	ELSIF (#coordSystem = "CS_MCS" AND #startPositionCoordSystem <> "CS_MCS")
	  OR (#coordSystem = "CS_JCS" AND #startPositionCoordSystem <> "CS_JCS")
	THEN
	  // Transform cartesian lastPos to MCS or JCS
	  #inverseKinematicsTransformation(AxesGroup         := #toKinematics,
	                                   Enable            := TRUE,
	                                   Position          := #statStartPosition,
	                                   CoordSystem       := #startPositionCoordSystem,
	                                   AxesCoordSystem   := #coordSystem,
	                                   LinkConstellation := #startLinkConstellation,
	                                   ErrorId           => #tempRetVal,
	                                   AxesPosition      => #statStartPosition);
	  
	  // check for error in last position calculation
	  IF #tempRetVal <> 16#0 THEN
	    #status := #tempRetVal;
	    RETURN;
	  END_IF;
	  
	ELSIF (#coordSystem <> "CS_MCS" AND #startPositionCoordSystem = "CS_MCS")
	  OR (#coordSystem <> "CS_JCS" AND #startPositionCoordSystem = "CS_JCS")
	THEN
	  // Transform axial lastPos to target cartesian CS
	  #kinematicsTransformation(AxesGroup         := #toKinematics,
	                            Enable            := TRUE,
	                            AxesPosition      := #statStartPosition,
	                            CoordSystem       := #coordSystem,
	                            AxesCoordSystem   := #startPositionCoordSystem,
	                            ErrorId           => #tempRetVal,
	                            Position          => #statStartPosition,
	                            LinkConstellation => #resultingLinkConstellation);
	  
	  // check for error in last position calculation
	  IF #tempRetVal <> 16#0 THEN
	    #status := #tempRetVal;
	    RETURN;
	  END_IF;
	  
	ELSE
	  // Transform Start position to correct CS 
	  "LKinCtrl_FrameTrans"(coordSystem    := #coordSystem, // Actual/Target CS
	                        coordSystemOld := #startPositionCoordSystem, // Last CS
	                        OCSFrames      := #OCSFrames, // OCS frames
	                        userFrames     := #userFrames,
	                        position       := #statStartPosition); // Position to be transformed
	END_IF;
	
	
	//------------------------------------------------------------------------------------------
	// Update linkConstellation
	//------------------------------------------------------------------------------------------
	// LinkConstellation can only be set at sPTP command in WCS/OCS
	IF #coordSystem <> "CS_MCS"
	  AND #coordSystem <> "CS_JCS"
	  AND #moveDirectParameter.linkConstellation <> 16#FFFF_FFFF
	  AND (#cmdType = "LKINCTRL_MC_MOVEDIRECTABS"
	  OR #cmdType = "LKINCTRL_MC_MOVEDIRECTREL")
	THEN
	  // LinkConstellation is changed
	  #resultingLinkConstellation := DWORD_TO_DINT(#moveDirectParameter.linkConstellation);
	END_IF;
	
	//------------------------------------------------------------------------------------------
	// Update PositionMode
	//------------------------------------------------------------------------------------------
	// PositionMode is only valid for absolute SPTP command in WCS/OCS
	IF #coordSystem <> "CS_MCS"
	  AND #moveDirectParameter.positionMode = "PM_ABS_REL" // Relative A coordinate
	  AND #cmdType = "LKINCTRL_MC_MOVEDIRECTABS"
	THEN
	  // Calc correct orientation position
	    #resultingPosition[4] := #statStartPosition[4] + #statCommandPosition[4];
	  //#statCommandPosition[4] := #resultingPosition[4]; // update tempPosition
	    ;
	END_IF;
	
	//------------------------------------------------------------------------------------------
	// ParameterValid bit check -> Check if all positions are valid -> LKinLang mechanism
	//------------------------------------------------------------------------------------------
	CASE #cmdType OF
	  "LKINCTRL_MC_MOVELINEARABS", "LKINCTRL_MC_MOVECIRCULARABS", "LKINCTRL_MC_MOVEDIRECTABS", "LKINCTRL_MC_MOVELINEARPICKANDPLACE":  // Absolute commands
	    FOR #tempIndex := 1 TO "LKINCTRL_NO_OF_VALID_BITS" DO
	      // Check valid bits and copy last pos (X,Y,Z,A) where missing
	      IF #parameterValid[#tempIndex] = FALSE THEN
	        #statCommandPosition[#tempIndex] := #statStartPosition[#tempIndex]; // write lastPos as target pos if invalid
	      ELSE
	        CONTINUE;
	      END_IF;
	    END_FOR;
	    
	  "LKINCTRL_MC_MOVELINEARREL", "LKINCTRL_MC_MOVECIRCULARREL", "LKINCTRL_MC_MOVEDIRECTREL":  // Relative commands
	    FOR #tempIndex := 1 TO "LKINCTRL_NO_OF_VALID_BITS" DO
	      // Check valid bits and set absolute pos to 0.0 (X,Y,Z,A)
	      IF #parameterValid[#tempIndex] = FALSE THEN
	        #statCommandPosition[#tempIndex] := 0.0; // write no increment as relative target pos if invalid
	      ELSE
	        CONTINUE;
	      END_IF;
	    END_FOR;
	    
	  ELSE  // Nothing to do for this cmdType
	    ;
	END_CASE;
	
	//------------------------------------------------------------------------------------------
	// Convert circle mode 3 (Gcode notation) to circle mode 1 (arc + endPoint)
	//------------------------------------------------------------------------------------------
	// --> CmdType = 3 (always absolute as result)
	// --> CircleParameters = calculated arc, updated auxPoint, circMode 1
	IF #circleParameters.circMode = "LKINCTRL_CIRCMODE_GCODE" THEN
	  #tempRetVal := "LKinCtrl_ConvCircMode3To1"(coordinates := #statCommandPosition,
	                                             startPosition := #statStartPosition,
	                                             cmdType := #cmdType,
	                                             circleParameters := #circleParameters);
	  
	  // check for error in circle calculation
	  IF #tempRetVal <> 16#0 THEN
	    #status := #tempRetVal;
	    RETURN;
	  END_IF;
	END_IF;
	
	//------------------------------------------------------------------------------------------
	// Handle relative shift
	//------------------------------------------------------------------------------------------
	IF #relativeShift.shiftActive = TRUE
	  AND #relativeShift.coordinateSystem = #coordSystem
	THEN
	  IF #cmdType = "LKINCTRL_MC_MOVELINEARABS"
	    OR #cmdType = "LKINCTRL_MC_MOVEDIRECTABS"
	    OR #cmdType = "LKINCTRL_MC_MOVECIRCULARABS"
	    OR #cmdType = "LKINCTRL_MC_MOVELINEARPICKANDPLACE"
	  THEN
	    // Translation and rotation (end point)
	    "LKinCtrl_OcsToWcs"(ocsX      := #relativeShift.coordinates[1],
	                        ocsY      := #relativeShift.coordinates[2],
	                        ocsZ      := #relativeShift.coordinates[3],
	                        ocsA      := #relativeShift.coordinates[4],
	                        ocsB      := #relativeShift.coordinates[5],
	                        ocsC      := #relativeShift.coordinates[6],
	                        pointXOcs := #statCommandPosition[1],
	                        pointYOcs := #statCommandPosition[2],
	                        pointZOcs := #statCommandPosition[3],
	                        pointAOcs := #statCommandPosition[4],
	                        pointBOcs := #statCommandPosition[5],
	                        pointCOcs := #statCommandPosition[6],
	                        pointXWcs => #statCommandPosition[1],
	                        pointYWcs => #statCommandPosition[2],
	                        pointZWcs => #statCommandPosition[3],
	                        pointAWcs => #statCommandPosition[4],
	                        pointBWcs => #statCommandPosition[5],
	                        pointCWcs => #statCommandPosition[6]);
	    
	    // Translation and rotation (aux point)
	    "LKinCtrl_OcsToWcs"(ocsX      := #relativeShift.coordinates[1],
	                        ocsY      := #relativeShift.coordinates[2],
	                        ocsZ      := #relativeShift.coordinates[3],
	                        ocsA      := #relativeShift.coordinates[4],
	                        ocsB      := #relativeShift.coordinates[5],
	                        ocsC      := #relativeShift.coordinates[6],
	                        pointXOcs := #circleParameters.auxPoint[1],
	                        pointYOcs := #circleParameters.auxPoint[2],
	                        pointZOcs := #circleParameters.auxPoint[3],
	                        pointAOcs := 0.0,
	                        pointBOcs := 0.0,
	                        pointCOcs := 0.0,
	                        pointXWcs => #circleParameters.auxPoint[1],
	                        pointYWcs => #circleParameters.auxPoint[2],
	                        pointZWcs => #circleParameters.auxPoint[3],
	                        pointAWcs => #tempAuxPoint[4],
	                        pointBWcs => #tempAuxPoint[5],
	                        pointCWcs => #tempAuxPoint[6]);
	    
	  ELSIF #cmdType = "LKINCTRL_MC_MOVELINEARREL"
	    OR #cmdType = "LKINCTRL_MC_MOVEDIRECTREL"
	    OR #cmdType = "LKINCTRL_MC_MOVECIRCULARREL"
	  THEN
	    // Only rotation (end point)
	    "LKinCtrl_OcsToWcs"(ocsX      := 0.0,
	                        ocsY      := 0.0,
	                        ocsZ      := 0.0,
	                        ocsA      := #relativeShift.coordinates[4],
	                        ocsB      := #relativeShift.coordinates[5],
	                        ocsC      := #relativeShift.coordinates[6],
	                        pointXOcs := #statCommandPosition[1],
	                        pointYOcs := #statCommandPosition[2],
	                        pointZOcs := #statCommandPosition[3],
	                        pointAOcs := 0.0,
	                        pointBOcs := 0.0,
	                        pointCOcs := 0.0,
	                        pointXWcs => #statCommandPosition[1],
	                        pointYWcs => #statCommandPosition[2],
	                        pointZWcs => #statCommandPosition[3],
	                        pointAWcs => #tempAuxPoint[4],
	                        pointBWcs => #tempAuxPoint[5],
	                        pointCWcs => #tempAuxPoint[6]);
	    
	    // Only rotation (aux point)
	    "LKinCtrl_OcsToWcs"(ocsX      := 0.0,
	                        ocsY      := 0.0,
	                        ocsZ      := 0.0,
	                        ocsA      := #relativeShift.coordinates[4],
	                        ocsB      := #relativeShift.coordinates[5],
	                        ocsC      := #relativeShift.coordinates[6],
	                        pointXOcs := #circleParameters.auxPoint[1],
	                        pointYOcs := #circleParameters.auxPoint[2],
	                        pointZOcs := #circleParameters.auxPoint[3],
	                        pointAOcs := 0.0,
	                        pointBOcs := 0.0,
	                        pointCOcs := 0.0,
	                        pointXWcs => #circleParameters.auxPoint[1],
	                        pointYWcs => #circleParameters.auxPoint[2],
	                        pointZWcs => #circleParameters.auxPoint[3],
	                        pointAWcs => #tempAuxPoint[4],
	                        pointBWcs => #tempAuxPoint[5],
	                        pointCWcs => #tempAuxPoint[6]);
	  ELSE
	    ;// No calculation necessary
	  END_IF;
	END_IF;
	
	//------------------------------------------------------------------------------------------
	// Calculate resulting absoulte position
	//------------------------------------------------------------------------------------------
	#tempRetVal := "LKinCtrl_CalcResultingPos"(cmdType := #cmdType,
	                                           cartesianPos := #statCommandPosition,
	                                           circleParameters := #circleParameters,
	                                           startPosition := #statStartPosition,
	                                           commandLengthIsZero => #cmdLengthZero,
	                                           resultingDistance => #resultingDistance,
	                                           resultingPosition => #resultingPosition,
	                                           resultingAuxPoint => #resultingAuxPoint);  
	
	// check for error in resulting position calculation
	IF #tempRetVal <> 16#0 THEN
	  #status := #tempRetVal;
	  RETURN;
	END_IF;
	
	//------------------------------------------------------------------------------------------
	// Transform UCS commands into WCS
	// At this point all coordinates are calauclated in UCS -> Transform them in WCS to be able to execute system commands
	//------------------------------------------------------------------------------------------
	IF #coordSystem >= "LKINCTRL_CS_NO_OF_FIRST_USER_FRAME"
	  AND #coordSystem <= "LKINCTRL_CS_NO_OF_LAST_USER_FRAME"
	THEN
	  CASE #cmdType OF
	    "LKINCTRL_MC_MOVELINEARABS", "LKINCTRL_MC_MOVECIRCULARABS", "LKINCTRL_MC_MOVEDIRECTABS",  // Absolute commands
	    "LKINCTRL_MC_MOVELINEARREL", "LKINCTRL_MC_MOVECIRCULARREL", "LKINCTRL_MC_MOVEDIRECTREL":  // Relative commands
	      // Up to this point all positions (start, resulting & distance) are in UCS
	      // --> Calculate new values in WCS
	      
	      // Transform start position into WCS
	      "LKinCtrl_OcsToWcs"(ocsX      := #userFrames[#coordSystem].x,
	                          ocsY      := #userFrames[#coordSystem].y,
	                          ocsZ      := #userFrames[#coordSystem].z,
	                          ocsA      := #userFrames[#coordSystem].a,
	                          ocsB      := #userFrames[#coordSystem].b,
	                          ocsC      := #userFrames[#coordSystem].c,
	                          pointXOcs := #statStartPosition[1],
	                          pointYOcs := #statStartPosition[2],
	                          pointZOcs := #statStartPosition[3],
	                          pointAOcs := #statStartPosition[4],
	                          pointBOcs := #statStartPosition[5],
	                          pointCOcs := #statStartPosition[6],
	                          pointXWcs => #statStartPosition[1],
	                          pointYWcs => #statStartPosition[2],
	                          pointZWcs => #statStartPosition[3],
	                          pointAWcs => #statStartPosition[4],
	                          pointBWcs => #statStartPosition[5],
	                          pointCWcs => #statStartPosition[6]);
	      
	      // Transform resulting position into WCS
	      "LKinCtrl_OcsToWcs"(ocsX      := #userFrames[#coordSystem].x,
	                          ocsY      := #userFrames[#coordSystem].y,
	                          ocsZ      := #userFrames[#coordSystem].z,
	                          ocsA      := #userFrames[#coordSystem].a,
	                          ocsB      := #userFrames[#coordSystem].b,
	                          ocsC      := #userFrames[#coordSystem].c,
	                          pointXOcs := #resultingPosition[1],
	                          pointYOcs := #resultingPosition[2],
	                          pointZOcs := #resultingPosition[3],
	                          pointAOcs := #resultingPosition[4],
	                          pointBOcs := #resultingPosition[5],
	                          pointCOcs := #resultingPosition[6],
	                          pointXWcs => #resultingPosition[1],
	                          pointYWcs => #resultingPosition[2],
	                          pointZWcs => #resultingPosition[3],
	                          pointAWcs => #resultingPosition[4],
	                          pointBWcs => #resultingPosition[5],
	                          pointCWcs => #resultingPosition[6]);
	      
	      // Transform resulting aux position into WCS
	      "LKinCtrl_OcsToWcs"(ocsX      := #userFrames[#coordSystem].x,
	                          ocsY      := #userFrames[#coordSystem].y,
	                          ocsZ      := #userFrames[#coordSystem].z,
	                          ocsA      := #userFrames[#coordSystem].a,
	                          ocsB      := #userFrames[#coordSystem].b,
	                          ocsC      := #userFrames[#coordSystem].c,
	                          pointXOcs := #resultingAuxPoint[1],
	                          pointYOcs := #resultingAuxPoint[2],
	                          pointZOcs := #resultingAuxPoint[3],
	                          pointAOcs := 0,
	                          pointBOcs := 0,
	                          pointCOcs := 0,
	                          pointXWcs => #resultingAuxPoint[1],
	                          pointYWcs => #resultingAuxPoint[2],
	                          pointZWcs => #resultingAuxPoint[3],
	                          pointAWcs => #tempAuxPoint[4],
	                          pointBWcs => #tempAuxPoint[5],
	                          pointCWcs => #tempAuxPoint[6]);
	      
	      // Calc resulting distance in WCS
	      FOR #tempIndex := 1 TO 6 DO
	        #resultingDistance[#tempIndex] := #resultingPosition[#tempIndex] - #statStartPosition[#tempIndex];
	      END_FOR;
	      
	      #coordSystem := "CS_WCS"; // Set CS to WCS
	  END_CASE;
	END_IF;
	
	
	
	
	
END_FUNCTION_BLOCK

FUNCTION "LKinCtrl_FrameTrans" : Void
TITLE = LKinCtrl_FrameTrans
{ S7_Optimized_Access := 'TRUE' }
AUTHOR : 'handling.team.automation@siemens.com'
FAMILY : LKinCtrl
VERSION : 5.0
//Transform postion into different coordinate systems
   VAR_INPUT 
      coordSystem : DInt;   // target coordinate system
      coordSystemOld : DInt;   // previous coordinate system
      OCSFrames : Array[1..3] of "LKinCtrl_typeFrame";   // OCS frames
      userFrames : Array["LKINCTRL_CS_NO_OF_FIRST_USER_FRAME".."LKINCTRL_CS_NO_OF_LAST_USER_FRAME"] of "LKinCtrl_typeFrame";   // User frames
   END_VAR

   VAR_IN_OUT 
      position : Array[1..6] of LReal;   // position to be transformed
   END_VAR


BEGIN
	//==========================================================================================
	// SIEMENS AG
	// (c)Copyright 2020 All Rights Reserved
	//------------------------------------------------------------------------------------------
	// Library: LKinCtrl
	// Tested with: S7-1517T-3 PN/DP
	// Engineering: TIA Portal V15
	// Restrictions: ---
	// Requirements: S7-1500T FW 2.5
	// Functionality: LKinCtrl_FrameTrans
	// The FC calculates a given position transformed into or from another coordinate system
	// depending on the actual / previous coordinate system of the cmd
	//
	// Support: tech.team.motioncontrol@siemens.com
	// Note: Parameter comments are only available in language 'English (United States)'
	//------------------------------------------------------------------------------------------
	// Change log table:
	// Version    Date          Expert in charge    Changes applied
	// 01.00.00   16.04.2019    JR                  First release version v1.0
	// 02.00.00   14.04.2020    FR                  Use array of frames
	// 03.00.00   18.01.2022    FR                  Update to 6 axis
	//===========================================================================================
	
	// Check if last CS differs from actual CS
	IF #coordSystem = #coordSystemOld THEN
	  // No calculation needed --> Return
	  RETURN;
	END_IF;
	
	// Calc new position
	// =================
	// Check if last CS was a OCS
	// YES: Transform position to WCS
	// NO: Do nothing --> Position is already in WCS
	CASE #coordSystemOld OF
	  "CS_OCS1".."CS_OCS3": // OCS
	    "LKinCtrl_OcsToWcs"(ocsX      := #OCSFrames[#coordSystemOld].x,
	                        ocsY      := #OCSFrames[#coordSystemOld].y,
	                        ocsZ      := #OCSFrames[#coordSystemOld].z,
	                        ocsA      := #OCSFrames[#coordSystemOld].a,
	                        ocsB      := #OCSFrames[#coordSystemOld].b,
	                        ocsC      := #OCSFrames[#coordSystemOld].c,
	                        pointXOcs := #position[1],
	                        pointYOcs := #position[2],
	                        pointZOcs := #position[3],
	                        pointAOcs := #position[4],
	                        pointBOcs := #position[5],
	                        pointCOcs := #position[6],
	                        pointXWcs => #position[1],
	                        pointYWcs => #position[2],
	                        pointZWcs => #position[3],
	                        pointAWcs => #position[4],
	                        pointBWcs => #position[5],
	                        pointCWcs => #position[6]);
	    
	  "LKINCTRL_CS_NO_OF_FIRST_USER_FRAME".."LKINCTRL_CS_NO_OF_LAST_USER_FRAME":  // User frame
	    "LKinCtrl_OcsToWcs"(ocsX      := #userFrames[#coordSystemOld].x,
	                        ocsY      := #userFrames[#coordSystemOld].y,
	                        ocsZ      := #userFrames[#coordSystemOld].z,
	                        ocsA      := #userFrames[#coordSystemOld].a,
	                        ocsB      := #userFrames[#coordSystemOld].b,
	                        ocsC      := #userFrames[#coordSystemOld].c,
	                        pointXOcs := #position[1],
	                        pointYOcs := #position[2],
	                        pointZOcs := #position[3],
	                        pointAOcs := #position[4],
	                        pointBOcs := #position[5],
	                        pointCOcs := #position[6],
	                        pointXWcs => #position[1],
	                        pointYWcs => #position[2],
	                        pointZWcs => #position[3],
	                        pointAWcs => #position[4],
	                        pointBWcs => #position[5],
	                        pointCWcs => #position[6]);
	    
	  ELSE
	    ;
	END_CASE;
	
	
	// Check if target CS is a OCS
	// YES: Transform position to target OCS
	// NO: Target CS is WCS --> Position is already in WCS from above
	CASE #coordSystem OF
	  "CS_OCS1".."CS_OCS3": // OCS
	    "LKinCtrl_WcsToOcs"(ocsX      := #OCSFrames[#coordSystem].x,
	                        ocsY      := #OCSFrames[#coordSystem].y,
	                        ocsZ      := #OCSFrames[#coordSystem].z,
	                        ocsA      := #OCSFrames[#coordSystem].a,
	                        ocsB      := #OCSFrames[#coordSystem].b,
	                        ocsC      := #OCSFrames[#coordSystem].c,
	                        pointXWcs := #position[1],
	                        pointYWcs := #position[2],
	                        pointZWcs := #position[3],
	                        pointAWcs := #position[4],
	                        pointBWcs := #position[5],
	                        pointCWcs := #position[6],
	                        pointXOcs => #position[1],
	                        pointYOcs => #position[2],
	                        pointZOcs => #position[3],
	                        pointAOcs => #position[4],
	                        pointBOcs => #position[5],
	                        pointCOcs => #position[6]);
	    
	  "LKINCTRL_CS_NO_OF_FIRST_USER_FRAME".."LKINCTRL_CS_NO_OF_LAST_USER_FRAME":  // User frame
	    "LKinCtrl_WcsToOcs"(ocsX      := #userFrames[#coordSystem].x,
	                        ocsY      := #userFrames[#coordSystem].y,
	                        ocsZ      := #userFrames[#coordSystem].z,
	                        ocsA      := #userFrames[#coordSystem].a,
	                        ocsB      := #userFrames[#coordSystem].b,
	                        ocsC      := #userFrames[#coordSystem].c,
	                        pointXWcs := #position[1],
	                        pointYWcs := #position[2],
	                        pointZWcs := #position[3],
	                        pointAWcs := #position[4],
	                        pointBWcs := #position[5],
	                        pointCWcs := #position[6],
	                        pointXOcs => #position[1],
	                        pointYOcs => #position[2],
	                        pointZOcs => #position[3],
	                        pointAOcs => #position[4],
	                        pointBOcs => #position[5],
	                        pointCOcs => #position[6]);
	    
	  ELSE
	    ;
	END_CASE;
	
	
	
END_FUNCTION

FUNCTION "LKinCtrl_ConvCircMode3To1" : Word
TITLE = LKinCtrl_ConvCircMode3To1
{ S7_Optimized_Access := 'TRUE' }
AUTHOR : 'handling.team.automation@siemens.com'
FAMILY : LKinCtrl
VERSION : 5.0
//The FC converts a circular motion command programmed with circMode 3 (GCode) to a circular command programmed with circMode 1 (center point and arc given)
   VAR_INPUT 
      coordinates : Array[1..6] of LReal;   // endPoint from path data element
      startPosition : Array[1..6] of LReal;
   END_VAR

   VAR_IN_OUT 
      cmdType : Int;   // cmdType of path data element
      circleParameters : "LKinCtrl_typeCircleParameters";   // circle parameters of path data element
   END_VAR

   VAR_TEMP 
      tempAuxPoint : Array[1..3] of LReal;   // resulting auxPoint
      tempEndPointResult : Array[1..6] of LReal;   // resulting endPoint
      tempOM : Array[1..2] of LReal;   // temporary math variable
      tempMS : Array[1..2] of LReal;   // temporary math variable
      tempME : Array[1..2] of LReal;   // temporary math variable
      tempAxisVector : Array[1..2] of LReal;   // temporary math variable
      tempScalarProd_ME_Axis : LReal;   // temporary math variable
      tempScalarProd_MS_Axis : LReal;   // temporary math variable
      tempLength_ME : LReal;   // temporary math variable
      tempLength_MS : LReal;   // temporary math variable
      tempAngleME_rad : LReal;   // temporary math variable
      tempAngleMS_rad : LReal;   // temporary math variable
      tempAngleME_deg : LReal;   // temporary math variable
      tempAngleMS_deg : LReal;   // temporary math variable
      tempAngleDiff_deg : LReal;   // temporary math variable
      tempCtr : Int;   // temporary counter
      tempCoordinates : Array[1..6] of LReal;   // temporary array for input end point
   END_VAR

   VAR CONSTANT 
      ARC_TOLERANCE : LReal := 1.0E-09;   // Tolerance when deciding arc
      RADIUS_TOLERANCE : LReal := 0.1;   // Tolerance when comparing calculated radius
      ERR_INVALID_RADIUS : Word := 16#8201;   // Error calculated radius is invalid
   END_VAR


BEGIN
	//==========================================================================================
	// SIEMENS AG
	// (c)Copyright 2020 All Rights Reserved
	//------------------------------------------------------------------------------------------
	// Library: LKinCtrl
	// Tested with: S7-1517T-3 PN/DP
	// Engineering: TIA Portal V15
	// Restrictions: ---
	// Requirements: S7-1500T FW 2.5
	// Functionality: LKinCtrl_ConvCircMode3To1
	// The FC converts a circular motion command programmed with circMode 3 (GCode) to a circular
	// command programmed with circMode 1 (center point and arc given)
	//
	// Support: tech.team.motioncontrol@siemens.com
	// Note: Parameter comments are only available in language 'English (United States)'
	//------------------------------------------------------------------------------------------
	// Change log table:
	// Version    Date          Expert in charge    Changes applied
	// 01.00.00   03.07.2019    JR                  First release version v1.0
	// 02.00.00   06.04.2020    FR                  Changed interface to fit PathDataPreBuf and normal element
	// 02.00.01   14.01.2021    FR                  Added tolerance when calculating arc
	// 02.00.02   19.10.2021    FR                  Changed check for ACOS to allow 0.0
	// 03.00.00   18.01.2022    FR                  Update to 6 axis; Check radius for plausability
	//===========================================================================================
	
	// Init retrun value
	#LKinCtrl_ConvCircMode3To1 := 16#0;
	
	// add conversion of circMode CM: 3 circular cmds -> CM: 1
	IF (#cmdType = "LKINCTRL_MC_MOVECIRCULARABS" OR #cmdType = "LKINCTRL_MC_MOVECIRCULARREL")
	  AND #circleParameters.circMode = "LKINCTRL_CIRCMODE_GCODE"
	THEN
	  // Copy input
	  #tempCoordinates := #coordinates;
	  
	  // conversion relative to absoulte for auxPoint (and EndPoint)
	  FOR #tempCtr := 1 TO 3 DO
	    // always convert auxPoint ==> always relative in this circle definition
	    #tempAuxPoint[#tempCtr] := #startPosition[#tempCtr] + #circleParameters.auxPoint[#tempCtr];// add new auxPoint as incremental value to last position
	    #circleParameters.auxPoint[#tempCtr] := #tempAuxPoint[#tempCtr]; // copy edited auxPoint to command for later use
	  END_FOR;
	  
	  // only convert endPoint in case of relative command
	  IF #cmdType = "LKINCTRL_MC_MOVECIRCULARREL" THEN
	    #tempEndPointResult[1] := #startPosition[1] + #tempCoordinates[1];
	    #tempEndPointResult[2] := #startPosition[2] + #tempCoordinates[2];
	    #tempEndPointResult[3] := #startPosition[3] + #tempCoordinates[3];
	    #tempEndPointResult[4] := #startPosition[4] + #tempCoordinates[4];
	    #tempEndPointResult[5] := #startPosition[5] + #tempCoordinates[5];
	    #tempEndPointResult[6] := #startPosition[6] + #tempCoordinates[6];
	    #cmdType := "LKINCTRL_MC_MOVECIRCULARABS";
	  ELSE
	    #tempEndPointResult := #tempCoordinates;
	  END_IF;
	  
	  // change circMode = 3 (define center and endPoint) to circMode = 1 (define center and arc)
	  #circleParameters.circMode := "CM_CENTER";
	  
	  // ----------------------------------------------------------------
	  // different behavior for different circlePlanes - write input vectors to calc variables 2D
	  // ----------------------------------------------------------------
	  // 0: ciclePlane XZ
	  IF #circleParameters.circlePlane = "CP_XZ" THEN
	    
	    // vector origin to circle center point 
	    #tempOM[1] := #tempAuxPoint[1];
	    #tempOM[2] := #tempAuxPoint[3];
	    
	    // unit vector x axis
	    #tempAxisVector[1] := 1;
	    #tempAxisVector[2] := 0;
	    
	    // vector circle center point to start point
	    #tempMS[1] := #startPosition[1] - #tempOM[1];
	    #tempMS[2] := #tempOM[2] - #startPosition[3];
	    
	    // vector circle center point to end point
	    #tempME[1] := #tempEndPointResult[1] - #tempOM[1];
	    #tempME[2] := #tempOM[2] - #tempEndPointResult[3];
	    
	    // 1: ciclePlane YZ
	  ELSIF #circleParameters.circlePlane = "CP_YZ" THEN
	    
	    // vector origin to circle center point 
	    #tempOM[1] := #tempAuxPoint[2];
	    #tempOM[2] := #tempAuxPoint[3];
	    
	    // unit vector x axis ==> simulating y axis here due to moved commands
	    #tempAxisVector[1] := 1;
	    #tempAxisVector[2] := 0;
	    
	    // vector circle center point to start point
	    #tempMS[1] := #startPosition[2] - #tempOM[1];
	    #tempMS[2] := #startPosition[3] - #tempOM[2];
	    
	    // vector circle center point to end point
	    #tempME[1] := #tempEndPointResult[2] - #tempOM[1];
	    #tempME[2] := #tempEndPointResult[3] - #tempOM[2];
	    
	    // 2: ciclePlane XY
	  ELSIF #circleParameters.circlePlane = "CP_XY" THEN
	    
	    // vector origin to circle center point 
	    #tempOM[1] := #tempAuxPoint[1];
	    #tempOM[2] := #tempAuxPoint[2];
	    
	    // unit vector x axis
	    #tempAxisVector[1] := 1;
	    #tempAxisVector[2] := 0;
	    
	    
	    // vector circle center point to start point
	    #tempMS[1] := #startPosition[1] - #tempOM[1];
	    #tempMS[2] := #startPosition[2] - #tempOM[2];
	    
	    // vector circle center point to end point
	    #tempME[1] := #tempEndPointResult[1] - #tempOM[1];
	    #tempME[2] := #tempEndPointResult[2] - #tempOM[2];
	    
	  ELSE
	    // error ==> wrong circlePlane
	    ;
	  END_IF;
	  
	  // ----------------------------------------------------------------
	  // VECTOR CALCULATIONS
	  // ----------------------------------------------------------------
	  // calc scalar product of ME (circle center point to end point) with x axis
	  #tempScalarProd_ME_Axis := "LKinCtrl_VecScalarProd_2D"(vIn1 := #tempME, vIn2 := #tempAxisVector);
	  // calc scalar product of MS (circle center point to start point / LastPos) with x axis
	  #tempScalarProd_MS_Axis := "LKinCtrl_VecScalarProd_2D"(vIn1 := #tempMS, vIn2 := #tempAxisVector);
	  
	  // calc vector length ME
	  #tempLength_ME := "LKinCtrl_VecAbs_2D"(#tempME);
	  // calc vector length MS
	  #tempLength_MS := "LKinCtrl_VecAbs_2D"(#tempMS);
	  
	  // Check if both radius are equal
	  IF ABS(#tempLength_ME - #tempLength_MS) > #RADIUS_TOLERANCE THEN
	    #LKinCtrl_ConvCircMode3To1 := #ERR_INVALID_RADIUS;
	    RETURN;
	  END_IF;
	  
	  // calc angle ME to axis
	  #tempAngleME_rad := ACOS(#tempScalarProd_ME_Axis / (#tempLength_ME * 1));
	  
	  IF #tempME[2] < 0 THEN
	    // invert angle due to ACOS range (only 0..PI)
	    #tempAngleME_rad := 2 * "LKINCTRL_PI" - #tempAngleME_rad;
	  ELSE
	    ;
	  END_IF;
	  // convert to degrees
	  #tempAngleME_deg := #tempAngleME_rad * 180 / "LKINCTRL_PI";
	  
	  // calc angle MS to axis
	  #tempAngleMS_rad := ACOS(#tempScalarProd_MS_Axis / (#tempLength_MS * 1));
	  // check for vector Ms to point downwards (below ! (x) axis)
	  IF #tempMS[2] < 0 THEN
	    // invert angle due to ACOS range
	    #tempAngleMS_rad := 2 * "LKINCTRL_PI" - #tempAngleMS_rad;
	  ELSE
	    ;
	  END_IF;
	  // convert to degrees
	  #tempAngleMS_deg := #tempAngleMS_rad * 180 / "LKINCTRL_PI";
	  
	  
	  // ----------------------------------------------------------------
	  // separation of path choice for angle calculation
	  // ----------------------------------------------------------------
	  // 0: CCW - counterclockwise / mathematical positive angle
	  IF #circleParameters.pathChoice = "PC_POSITIVE" THEN
	    // calculate difference angle
	    #tempAngleDiff_deg := #tempAngleME_deg - #tempAngleMS_deg;
	    IF #tempAngleDiff_deg > #ARC_TOLERANCE THEN
	      // write caclulated angle
	      #circleParameters.arc := #tempAngleDiff_deg;
	    ELSE
	      // write caclulated angle ==> add 360 degrees to get positive angle value
	      #circleParameters.arc := #tempAngleDiff_deg + 360;
	    END_IF;
	    
	    // 1: CW - clockwise / mathematical negative angle
	  ELSIF #circleParameters.pathChoice = "PC_NEGATIVE" THEN
	    // calculate difference angle
	    #tempAngleDiff_deg := #tempAngleMS_deg - #tempAngleME_deg;
	    IF #tempAngleDiff_deg > #ARC_TOLERANCE THEN
	      // write caclulated angle
	      #circleParameters.arc := #tempAngleDiff_deg;
	    ELSE
	      // write caclulated angle ==> add 360 degrees to get positive angle value
	      #circleParameters.arc := #tempAngleDiff_deg + 360;
	    END_IF;
	    
	  ELSE
	    // wrong input for pathChoice
	    ;
	  END_IF;
	  
	ELSE
	  ;// nothing to do
	END_IF;
END_FUNCTION

FUNCTION "LKinCtrl_VecScalarProd_2D" : LReal
TITLE = LKinCtrl_VecScalarProd_2D
{ S7_Optimized_Access := 'TRUE' }
AUTHOR : 'handling.team.automation@siemens.com'
FAMILY : LKinCtrl
VERSION : 5.0
//Calculates the scalar product of given vectors
   VAR_INPUT 
      vIn1 : Array[1..2] of LReal;   // Input vector 1
      vIn2 : Array[1..2] of LReal;   // Input vector 2
   END_VAR


BEGIN
	//=============================================================================
	// SIEMENS AG
	// (c)Copyright 2019 All Rights Reserved
	//-----------------------------------------------------------------------------
	// Library: - 
	// Tested with: S7-1516T-3 PN
	// Engineering: TIA Portal V15
	// Restrictions: -
	// Requirements: S7-1500/S7-1500T FW 2.5
	// Functionality: Scalar product of two coordinates
	//-----------------------------------------------------------------------------
	// Change log table:
	// Version  Date       Expert in charge Changes applied
	// 01.00.00 27.08.2018 SF               created
	// 01.00.01 29.01.2019 JR               adaptions for LKinCtrl 
	//=============================================================================
	
	#LKinCtrl_VecScalarProd_2D := (* #vIn1[0]*#vIn2[0] + *)#vIn1[1] * #vIn2[1] + #vIn1[2] * #vIn2[2];
END_FUNCTION

FUNCTION "LKinCtrl_VecAbs_2D" : LReal
TITLE = LKinCtrl_VecAbs_2D
{ S7_Optimized_Access := 'TRUE' }
AUTHOR : 'handling.team.automation@siemens.com'
FAMILY : LKinCtrl
VERSION : 5.0
//Calculates the length of a given vector in 2D
   VAR_INPUT 
      vIn : Array[1..2] of LReal;   // Input vector
   END_VAR


BEGIN
	//=============================================================================
	// SIEMENS AG
	// (c)Copyright 2019 All Rights Reserved
	//-----------------------------------------------------------------------------
	// Library: - 
	// Tested with: S7-1516T-3 PN
	// Engineering: TIA Portal V15
	// Restrictions: -
	// Requirements: S7-1500/S7-1500T FW 2.5
	// Functionality: Calculate length of vector
	//-----------------------------------------------------------------------------
	// Change log table:
	// Version  Date       Expert in charge Changes applied
	// 01.00.00 27.08.2018 SF               created
	// 01.00.01 29.01.2019 JR               adaptions for LKinCtrl 
	//=============================================================================
	
	#LKinCtrl_VecAbs_2D := SQRT((* #vIn[0]*#vIn[0] + *)#vIn[1] * #vIn[1] + #vIn[2] * #vIn[2]);
END_FUNCTION

FUNCTION "LKinCtrl_CalcResultingPos" : Word
TITLE = LKinCtrl_CalcResultingPos
{ S7_Optimized_Access := 'TRUE' }
AUTHOR : 'handling.team.automation@siemens.com'
FAMILY : LKinCtrl
VERSION : 5.0
//The FC calculates the resulting last position after a given command being executed starting from a given 'previous' last position 
   VAR_INPUT 
      cmdType : Int;   // command type
      cartesianPos : Array[1..6] of LReal;   // cartesian position (target from command)
      circleParameters : "LKinCtrl_typeCircleParameters";   // circle parameters
      startPosition : Array[1..6] of LReal;   // start of command (last target position)
   END_VAR

   VAR_OUTPUT 
      commandLengthIsZero : Bool;   // TRUE: command has a length of 0.0; FALSE: Command has a length
      resultingPosition : Array[1..6] of LReal;   // resulting last position
      resultingDistance : Array[1..6] of LReal;   // distance between start and endpoint for relative commands
      resultingAuxPoint : Array[1..3] of LReal;   // resulting auxPoint
   END_VAR

   VAR_TEMP 
      tempIndex : Int;   // temporary counter
      tempCartesianPos : Array[1..6] of LReal;   // temporary copy of cartesian position (target from command)
      tempResultingAuxPoint : Array[1..3] of LReal;   // temporary resulting auxPoint
   END_VAR

   VAR CONSTANT 
      STATUS_NO_ERROR : Word := 16#0000;   // status no error occured
   END_VAR


BEGIN
	//==========================================================================================
	// SIEMENS AG
	// (c)Copyright 2020 All Rights Reserved
	//------------------------------------------------------------------------------------------
	// Library: LKinCtrl
	// Tested with: S7-1517T-3 PN/DP
	// Engineering: TIA Portal V16
	// Restrictions: ---
	// Requirements: S7-1500T FW 2.8
	// Functionality: LKinCtrl_CalcResultingPos
	// The FC calculates the resulting last position after a given command being executed
	// starting from a given 'previous' last position 
	//
	// Support: tech.team.motioncontrol@siemens.com
	// Note: Parameter comments are only available in language 'English (United States)'
	//------------------------------------------------------------------------------------------
	// Change log table:
	// Version    Date          Expert in charge    Changes applied
	// 01.00.00   11.03.2019    JR                  First release version v1.0
	// 01.00.01   17.05.2019    JR                  formal code changes fitting to styleguide
	// 02.00.00   06.04.2020    FR                  Changed interface to fit PathDataPreBuf and normal element; Also updated the calculation
	// 02.01.00   16.04.2020    FR                  Added moveDirect
	// 03.00.00   25.01.2021    FR                  Changed interface and rework
	// 04.00.00   18.01.2022    FR                  Update to 6 axis, added distance
	// 04.01.00   16.10.2023    AH                  Added relative shift
	// 04.01.00   09.01.2024    SF                  Added PickAndPlace command#
	// 04.01.01   25.04.2024    JH                  Bugfix for uninitialized output
	// 04.02.00   11.07.2024    AH                  Fixed wrong calculation of circularCommand in UCS
	//===========================================================================================
	
	// ---------------------------------------------------------
	// Initialize return value to no error
	// ---------------------------------------------------------
	#LKinCtrl_CalcResultingPos := #STATUS_NO_ERROR;
	#commandLengthIsZero := FALSE;
	
	// ---------------------------------------------------------
	// Copy input position to temp
	// ---------------------------------------------------------
	#tempCartesianPos := #cartesianPos;
	
	// Reset distance output
	FOR #tempIndex := 1 TO 6 DO
	    #resultingDistance[#tempIndex] := 0.0;
	END_FOR;
	
	// ---------------------------------------------------------
	// Check if command has length 0.0 --> Nothing to calculate
	// ---------------------------------------------------------
	CASE #cmdType OF
	    "LKINCTRL_MC_MOVELINEARABS", "LKINCTRL_MC_MOVEDIRECTABS":
	        // Check all coordinates to be last position
	        FOR #tempIndex := 1 TO 6 DO
	            IF #tempCartesianPos[#tempIndex] = #startPosition[#tempIndex] THEN
	                #commandLengthIsZero := TRUE;
	            ELSE
	                #commandLengthIsZero := FALSE;
	                EXIT;
	            END_IF;
	        END_FOR;
	        
	    "LKINCTRL_MC_MOVELINEARREL", "LKINCTRL_MC_MOVEDIRECTREL":
	        // Check all coordinates to be 0.0
	        FOR #tempIndex := 1 TO 6 DO
	            IF #tempCartesianPos[#tempIndex] = 0.0 THEN
	                #commandLengthIsZero := TRUE;
	            ELSE
	                #commandLengthIsZero := FALSE;
	                EXIT;
	            END_IF;
	        END_FOR;
	        
	    "LKINCTRL_MC_MOVECIRCULARABS", "LKINCTRL_MC_MOVECIRCULARREL":
	        // Always calculate circular commands
	        #commandLengthIsZero := FALSE;
	        
	    "LKINCTRL_MC_MOVELINEARPICKANDPLACE":
	        // Check all coordinates to be last position
	        FOR #tempIndex := 1 TO 6 DO
	            IF #tempCartesianPos[#tempIndex] = #startPosition[#tempIndex] THEN
	                #commandLengthIsZero := TRUE;
	            ELSE
	                #commandLengthIsZero := FALSE;
	                EXIT;
	            END_IF;
	        END_FOR;
	        
	    "LKINCTRL_CMD_FLAG_ONLY",
	    "LKINCTRL_MC_TRACKCONVEYORBELT",
	    "LKINCTRL_MC_SET_OCS_FRAME",
	    "LKINCTRL_MC_SET_USER_FRAME",
	    "LKINCTRL_MC_SHIFT_CS_REL",               //added relative shift + reset
	    "LKINCTRL_MC_RESET_SHIFT",
	    "LKINCTRL_MC_ACTIVATE_TOOL",
	    "LKINCTRL_MC_SET_TOOL_FRAME",
	    "LKINCTRL_MC_DEFINE_WS_ZONE",
	    "LKINCTRL_MC_ACTIVATE_WS_ZONE",
	    "LKINCTRL_MC_DEACTIVATE_WS_ZONE",
	    "LKINCTRL_MC_DEFINE_KIN_ZONE",
	    "LKINCTRL_MC_ACTIVATE_KIN_ZONE",
	    "LKINCTRL_MC_DEACTIVATE_KIN_ZONE",
	    "LKINCTRL_CONFIG_END_OFFSET_COMP",
	    "LKINCTRL_CONFIG_START_OFFSET_COMP_LEFT",
	    "LKINCTRL_CONFIG_START_OFFSET_COMP_RIGHT",
	    "LKINCTRL_CMD_WAIT_TIME",
	    "LKINCTRL_MC_DESYNC_CONVEYOR":
	        // All configuration commands or other
	        #commandLengthIsZero := TRUE;
	        
	    ELSE
	        
	        #commandLengthIsZero := FALSE;
	END_CASE;
	
	// ---------------------------------------------------------
	// Check if length of command is 0.0 -> Skip calculation and return
	// ---------------------------------------------------------
	IF #commandLengthIsZero = TRUE THEN
	    #resultingPosition := #startPosition;
	    FOR #tempIndex := 1 TO 6 DO
	        #resultingDistance[#tempIndex] := 0.0;
	    END_FOR;
	    RETURN;
	END_IF;
	
	// ---------------------------------------------------------
	// Calculate resulting position and auxPoint
	// ---------------------------------------------------------
	CASE #cmdType OF
	    "LKINCTRL_MC_MOVELINEARABS", "LKINCTRL_MC_MOVEDIRECTABS", "LKINCTRL_MC_MOVELINEARPICKANDPLACE":  // Linear absolute & MoveDirect absolute
	        // Calculate resulting distance for linear absolute commands
	        FOR #tempIndex := 1 TO 6 DO
	            #resultingDistance[#tempIndex] := #tempCartesianPos[#tempIndex] - #startPosition[#tempIndex];
	        END_FOR;
	        #resultingPosition := #tempCartesianPos; // Directly copy given target position
	        
	    "LKINCTRL_MC_MOVELINEARREL", "LKINCTRL_MC_MOVEDIRECTREL": // Linear relative & MoveDirect relative
	        // Calculate resulting targetPosition for linear relative command
	        FOR #tempIndex := 1 TO 6 DO
	            #resultingPosition[#tempIndex] := #startPosition[#tempIndex] + #tempCartesianPos[#tempIndex];
	        END_FOR;
	        #resultingDistance := #tempCartesianPos;
	        
	    "LKINCTRL_MC_MOVECIRCULARABS":
	        CASE #circleParameters.circMode OF
	            "CM_BORDER", "LKINCTRL_CIRCMODE_GCODE": // CM 0 & 3
	                FOR #tempIndex := 1 TO 6 DO
	                    #resultingDistance[#tempIndex] := #tempCartesianPos[#tempIndex] - #startPosition[#tempIndex];
	                END_FOR;
	                
	                #resultingPosition := #tempCartesianPos; // directly copy given endPoint as LastPos
	                #tempResultingAuxPoint := #circleParameters.auxPoint; // directly copy given auxPoint
	                
	                
	            "CM_CENTER":  // CM 1
	                #tempResultingAuxPoint := #circleParameters.auxPoint; // directly copy given auxPoint
	                
	                // Calculate lastPos[1..3] from arc
	                #LKinCtrl_CalcResultingPos := "LKinCtrl_CalcPosFromAux"(arc := #circleParameters.arc,
	                                                                        circlePlane := #circleParameters.circlePlane,
	                                                                        pathChoice := #circleParameters.pathChoice,
	                                                                        auxPoint := #tempResultingAuxPoint,
	                                                                        startPosition := #startPosition,
	                                                                        endPosition => #resultingPosition);
	                
	                #resultingPosition[4] := #tempCartesianPos[4]; // Update orientation position
	                #resultingPosition[5] := #tempCartesianPos[5]; // Update orientation position
	                #resultingPosition[6] := #tempCartesianPos[6]; // Update orientation position
	                
	                IF #LKinCtrl_CalcResultingPos <> #STATUS_NO_ERROR THEN
	                    #resultingAuxPoint := #tempResultingAuxPoint;
	                    RETURN;
	                END_IF;
	                
	            "CM_RADIUS": // CM 2
	                FOR #tempIndex := 1 TO 6 DO
	                    #resultingDistance[#tempIndex] := #tempCartesianPos[#tempIndex] - #startPosition[#tempIndex];
	                END_FOR;
	                
	                // only write parameters for used planes ==> exclude unused plane coordinates for relative commands
	                IF #circleParameters.circlePlane = "CP_XZ" THEN   // XZ plane
	                    #resultingPosition[1] := #tempCartesianPos[1];
	                    // exclude y coordinate
	                    #resultingPosition[3] := #tempCartesianPos[3];
	                ELSIF #circleParameters.circlePlane = "CP_YZ" THEN   // YZ plane
	                    // exclude x coordinate
	                    #resultingPosition[2] := #tempCartesianPos[2];
	                    #resultingPosition[3] := #tempCartesianPos[3];
	                ELSIF #circleParameters.circlePlane = "CP_XY" THEN   // XY plane
	                    #resultingPosition[1] := #tempCartesianPos[1];
	                    #resultingPosition[2] := #tempCartesianPos[2];
	                    // exclude z coordinate
	                END_IF;
	                
	                // Always write orientation
	                #resultingPosition[4] := #tempCartesianPos[4];
	                #resultingPosition[5] := #tempCartesianPos[5];
	                #resultingPosition[6] := #tempCartesianPos[6];
	                
	                
	        END_CASE;
	        
	        
	    "LKINCTRL_MC_MOVECIRCULARREL":
	        CASE #circleParameters.circMode OF
	            "CM_BORDER", "LKINCTRL_CIRCMODE_GCODE": // CM 0 & 3
	                // Calculate absoulte AuxPoint first with starting point (last pos)
	                FOR #tempIndex := 1 TO 3 DO
	                    #tempResultingAuxPoint[#tempIndex] := #startPosition[#tempIndex] + #circleParameters.auxPoint[#tempIndex];
	                END_FOR;
	                // Calculate absoulte EndPoint after auxPoint -> lastPos is now endPoint
	                FOR #tempIndex := 1 TO 6 DO
	                    #resultingPosition[#tempIndex] := #startPosition[#tempIndex] + #tempCartesianPos[#tempIndex];
	                END_FOR;
	                
	                #resultingDistance := #tempCartesianPos;
	                
	                
	            "CM_CENTER":  // CM 1
	                // run same calculation to MC_MOVECIRCULARABS, but convert (rel -> abs) auxPoint before
	                FOR #tempIndex := 1 TO 3 DO
	                    #tempResultingAuxPoint[#tempIndex] := #startPosition[#tempIndex] + #circleParameters.auxPoint[#tempIndex];
	                END_FOR;
	                
	                // Calculate lastPos[1..3] from arc
	                #LKinCtrl_CalcResultingPos := "LKinCtrl_CalcPosFromAux"(arc := #circleParameters.arc,
	                                                                        circlePlane := #circleParameters.circlePlane,
	                                                                        pathChoice := #circleParameters.pathChoice,
	                                                                        auxPoint := #tempResultingAuxPoint,
	                                                                        startPosition := #startPosition,
	                                                                        endPosition => #resultingPosition);
	                
	                #resultingPosition[4] := #startPosition[4] + #tempCartesianPos[4]; // Update orientation position
	                #resultingPosition[5] := #startPosition[5] + #tempCartesianPos[5]; // Update orientation position
	                #resultingPosition[6] := #startPosition[6] + #tempCartesianPos[6]; // Update orientation position
	                
	                IF #LKinCtrl_CalcResultingPos <> #STATUS_NO_ERROR THEN
	                    #resultingAuxPoint := #tempResultingAuxPoint;
	                    RETURN;
	                END_IF;
	                
	            "CM_RADIUS": // CM 2
	                // only write parameters for used planes ==> exclude unused plane coordinates for relative commands
	                IF #circleParameters.circlePlane = "CP_XZ" THEN   // XZ plane
	                    #resultingPosition[1] := #startPosition[1] + #tempCartesianPos[1];
	                    // exclude y coordinate
	                    #resultingPosition[3] := #startPosition[3] + #tempCartesianPos[3];
	                ELSIF #circleParameters.circlePlane = "CP_YZ" THEN   // YZ plane
	                    // exclude x coordinate
	                    #resultingPosition[2] := #startPosition[2] + #tempCartesianPos[2];
	                    #resultingPosition[3] := #startPosition[3] + #tempCartesianPos[3];
	                ELSIF #circleParameters.circlePlane = "CP_XY" THEN   // XY plane
	                    #resultingPosition[1] := #startPosition[1] + #tempCartesianPos[1];
	                    #resultingPosition[2] := #startPosition[2] + #tempCartesianPos[2];
	                    // exclude z coordinate
	                END_IF;
	                // Always write orientation
	                #resultingPosition[4] := #startPosition[4] + #tempCartesianPos[4];
	                #resultingPosition[5] := #startPosition[5] + #tempCartesianPos[5];
	                #resultingPosition[6] := #startPosition[6] + #tempCartesianPos[6];
	                
	                #resultingDistance := #tempCartesianPos;
	        END_CASE;
	        
	    ELSE
	        // Other commands
	        ;
	END_CASE;
	
	// copy to output
	#resultingAuxPoint := #tempResultingAuxPoint;
	
	
	
END_FUNCTION

FUNCTION "LKinCtrl_CalcPosFromAux" : Word
TITLE = LKinCtrl_CalcPosFromAux
{ S7_Optimized_Access := 'TRUE' }
AUTHOR : 'handling.team.automation@siemens.com'
FAMILY : LKinCtrl
VERSION : 5.0
//Calculates the resulting position from and circular command with auxPoint and arc
   VAR_INPUT 
      arc : LReal;   // arc input
      circlePlane : DInt;   // circle plane input
      pathChoice : DInt;   // path choice input
      auxPoint : Array[1..3] of LReal;   // auxPoint input
      startPosition : Array[1..6] of LReal;   // start position input
   END_VAR

   VAR_OUTPUT 
      endPosition : Array[1..6] of LReal;   // resulting last position
   END_VAR

   VAR_TEMP 
      tempCircRadiusPt1 : LReal;   // temporary variable for calculation
      tempCircRadiusPt2 : LReal;   // temporary variable for calculation
      tempCircRadiusPt3 : LReal;   // temporary variable for calculation
      tempCircRadius : LReal;   // temporary variable for calculation
      tempCircleDirectionSign : Int;   // temporary variable for calculation
      tempAngleRadius : LReal;   // temporary variable for calculation
      tempArgAcos : LReal;   // temporary variable for calculation
      tempArc : LReal;   // temporary variable for arc
   END_VAR

   VAR CONSTANT 
      NO_ERROR : Word := 16#0000;   // no error
      ERR_INVALID_CIRCLEPLANE : Word := 16#8265;   // error due to invalid  circle plane
      ERR_INVALID_PATHCHOICE : Word := 16#8266;   // error due to invalid path choice
   END_VAR


BEGIN
	//==========================================================================================
	// SIEMENS AG
	// (c)Copyright 2021 All Rights Reserved
	//------------------------------------------------------------------------------------------
	// Library: LKinCtrl
	// Tested with: S7-1517T-3 PN/DP
	// Engineering: TIA Portal V16
	// Restrictions: ---
	// Requirements: S7-1500T FW 2.8
	// Functionality: LKinCtrl_CalcPosFromAux
	// The FC calculates the resulting position after a given command being executed
	// starting from a given 'previous' last position 
	//
	// Support: tech.team.motioncontrol@siemens.com
	// Note: Parameter comments are only available in language 'English (United States)'
	//------------------------------------------------------------------------------------------
	// Change log table:
	// Version    Date          Expert in charge    Changes applied
	// 01.00.00   05.02.2021    FR                  First released version
	// 04.02.00   11.07.2024    AH                  Fixed wrong calculation of circularCommand in UCS
	//===========================================================================================
	
	// Init return value
	#LKinCtrl_CalcPosFromAux := #NO_ERROR;
	
	// Copy arc to temp
	#tempArc := #arc;
	
	// check for angles bigger than full circle (360 degrees)
	IF #tempArc > 360.0 THEN
	    #tempArc := LREAL_TO_DINT(#tempArc) MOD 360; // check for angles being multiple of 360 degrees (system commands do run bigger circles)
	END_IF;
	
	// try catching complete circles without calculation
	IF #tempArc = 360.0 OR #tempArc = 0.0 THEN
	    RETURN; // keep old positions, do nothing
	END_IF;
	
	// calculate radius of circle around auxPoint - new 
	CASE #circlePlane OF
	    "CP_XZ":  // 0: "CP_XZ" - circle plane XZ
	        #tempCircRadiusPt1 := (#startPosition[1] - #auxPoint[1]) * (#startPosition[1] - #auxPoint[1]);
	        #tempCircRadiusPt2 := 0.0;//((lastPos[2] - lastAuxPoint[2]) * (lastPos[2] - lastAuxPoint[2]);
	        #tempCircRadiusPt3 := (#startPosition[3] - #auxPoint[3]) * (#startPosition[3] - #auxPoint[3]);
	    "CP_YZ":  // 1: "CP_YZ" - circle plane YZ
	        #tempCircRadiusPt1 := 0.0;//((lastPos[1] - lastAuxPoint[1]) * (lastPos[1] - lastAuxPoint[1]);
	        #tempCircRadiusPt2 := (#startPosition[2] - #auxPoint[2]) * (#startPosition[2] - #auxPoint[2]);
	        #tempCircRadiusPt3 := (#startPosition[3] - #auxPoint[3]) * (#startPosition[3] - #auxPoint[3]);
	    "CP_XY":  // 2: "CP_XY" - circle plane XY
	        #tempCircRadiusPt1 := (#startPosition[1] - #auxPoint[1]) * (#startPosition[1] - #auxPoint[1]);
	        #tempCircRadiusPt2 := (#startPosition[2] - #auxPoint[2]) * (#startPosition[2] - #auxPoint[2]);
	        #tempCircRadiusPt3 := 0.0;//(lastPos[3] - lastAuxPoint[3]) * (lastPos[3] - lastAuxPoint[3]);
	    ELSE
	        // wrong circle plane, error will be caught earlier when checking PathDataElement
	        #LKinCtrl_CalcPosFromAux := #ERR_INVALID_CIRCLEPLANE;
	        RETURN;
	END_CASE;
	
	// Calculate radius
	#tempCircRadius := SQRT_LREAL(#tempCircRadiusPt1 + #tempCircRadiusPt2 + #tempCircRadiusPt3);
	
	IF #tempCircRadius = 0.0 THEN
	    // Radius is 0.0 --> Not allowed
	    // #LKinCtrl_CalcPosFromAux := #ERR_RADIUS_ZERO;
	    RETURN;
	END_IF;
	
	// check for circleDirection -> define sign for motion command parameter 'arc'
	CASE #pathChoice OF
	    "PC_POSITIVE":  // 0: PC_Positive - positive direction (CCW)
	        #tempCircleDirectionSign := 1;
	    "PC_NEGATIVE":  // 1: PC_Negative - negative direction (CW)
	        #tempCircleDirectionSign := -1;
	    ELSE
	        // Wrong circle direction
	        #LKinCtrl_CalcPosFromAux := #ERR_INVALID_PATHCHOICE;
	        RETURN;
	END_CASE;
	
	// Init endposition with start
	#endPosition := #startPosition;
	
	// Calculate position
	CASE #circlePlane OF
	    "CP_XZ":  // 0: "CP_XZ" - circle plane XZ
	        // invert circle direction again --> See definition of XZ plane is actually ZX plane!
	        #tempCircleDirectionSign *= -1;
	        
	        // calculate argument for ACOS (angle in between of two vectors - radius and x axis)
	        #tempArgAcos := ((#startPosition[1] - #auxPoint[1]) * 1) / (#tempCircRadius * SQRT_LREAL(1));
	        // calculate ACOS for angle between to vectors
	        #tempAngleRadius := ACOS_LREAL(#tempArgAcos) * 180.0 / "LKINCTRL_PI";
	        
	        // check circle center point to be below (y direction) start point
	        IF #auxPoint[3] > #startPosition[3] THEN
	            #tempAngleRadius := #tempAngleRadius * -1; // acos result changed to negative angle
	        ELSIF #auxPoint[3] < #startPosition[3] THEN
	            #tempAngleRadius := #tempAngleRadius;
	        END_IF;
	        
	        #endPosition[1] := #tempCircRadius * COS_LREAL((#tempArc * #tempCircleDirectionSign + #tempAngleRadius) * "LKINCTRL_PI" / 180.0) + #auxPoint[1];
	        #endPosition[3] := #tempCircRadius * SIN_LREAL((#tempArc * #tempCircleDirectionSign + #tempAngleRadius) * "LKINCTRL_PI" / 180.0) + #auxPoint[3];
	        
	        
	    "CP_YZ":   // 1: "CP_YZ" - circle plane YZ
	        // calculate argument for ACOS (angle in between of two vectors - radius and x axis)
	        #tempArgAcos := ((#startPosition[2] - #auxPoint[2]) * 1) / (#tempCircRadius * SQRT_LREAL(1));
	        // calculate ACOS for angle between to vectors
	        #tempAngleRadius := ACOS_LREAL(#tempArgAcos) * 180.0 / "LKINCTRL_PI";
	        
	        // check circle center point to be below (y direction) start point
	        IF #auxPoint[3] > #startPosition[3] THEN
	            #tempAngleRadius := #tempAngleRadius * -1; // acos result changed to negative angle
	        ELSIF #auxPoint[3] < #startPosition[3] THEN
	            #tempAngleRadius := #tempAngleRadius;
	        END_IF;
	        
	        #endPosition[2] := #tempCircRadius * COS_LREAL((#tempArc * #tempCircleDirectionSign + #tempAngleRadius) * "LKINCTRL_PI" / 180.0) + #auxPoint[2];
	        #endPosition[3] := #tempCircRadius * SIN_LREAL((#tempArc * #tempCircleDirectionSign + #tempAngleRadius) * "LKINCTRL_PI" / 180.0) + #auxPoint[3];
	        
	        
	    "CP_XY":  // 2: "CP_XY" - circle plane XY
	        // calculate argument for ACOS (angle in between of two vectors - radius and x axis)
	        #tempArgAcos := ((#startPosition[1] - #auxPoint[1]) * 1) / (#tempCircRadius * SQRT_LREAL(1));
	        // calculate ACOS for angle between to vectors
	        #tempAngleRadius := ACOS_LREAL(#tempArgAcos) * 180.0 / "LKINCTRL_PI";
	        
	        // check circle center point to be below (y direction) start point
	        IF #auxPoint[2] > #startPosition[2] THEN
	            #tempAngleRadius := #tempAngleRadius * -1;// acos result changed to negative angle
	        ELSIF #auxPoint[2] < #startPosition[2] THEN // Changed > to < // FR 2019/04/17
	            #tempAngleRadius := #tempAngleRadius;
	        END_IF;
	        
	        #endPosition[1] := #tempCircRadius * COS_LREAL((#tempArc * #tempCircleDirectionSign + #tempAngleRadius) * "LKINCTRL_PI" / 180.0) + #auxPoint[1];
	        #endPosition[2] := #tempCircRadius * SIN_LREAL((#tempArc * #tempCircleDirectionSign + #tempAngleRadius) * "LKINCTRL_PI" / 180.0) + #auxPoint[2];
	    ELSE
	        // Wrong circle direction
	        #LKinCtrl_CalcPosFromAux := #ERR_INVALID_CIRCLEPLANE;
	        RETURN;
	END_CASE;
	
END_FUNCTION

FUNCTION "LKinCtrl_GetPathDataCmd" : Word
TITLE = LKinCtrl_GetPathDataCmd
{ S7_Optimized_Access := 'TRUE' }
AUTHOR : 'handling.team.automation@siemens.com'
FAMILY : LKinCtrl
VERSION : 5.0
//Copy the path command from any path data type at the given index
   VAR_INPUT 
      pathDataType : USInt;   // Type of path data which is connected
      index : DInt;   // Index to be copied
   END_VAR

   VAR_OUTPUT 
      pathDataCommand : "LKinCtrl_typePathDataElement";   // Resulting path data command
      parameterValid : Array[1.."LKINCTRL_NO_OF_VALID_BITS"] of Bool;   // Resulting parameter valid bits
   END_VAR

   VAR_IN_OUT 
      pathData : "LKinCtrl_typePathData";
      pointTable : Array[*] of "LKinCtrl_typePoint";   // Point table
   END_VAR

   VAR_TEMP 
      tempCtr : DInt;   // Temporary counter
      tempPoint : DInt;   // Temporary index of point in point table
   END_VAR


BEGIN
	//==========================================================================================
	// SIEMENS AG
	// (c)Copyright 2020 All Rights Reserved
	//------------------------------------------------------------------------------------------
	// Library: LKinCtrl
	// Tested with: S7-1517T-3 PN/DP
	// Engineering: TIA Portal V15
	// Restrictions: ---
	// Requirements: S7-1500T FW 2.5
	// Functionality: LKinCtrl_GetPathDataCmd
	// The FC copies the path data command at the given index to the output.
	//
	// Support: tech.team.motioncontrol@siemens.com
	// Note: Parameter comments are only available in language 'English (United States)'
	//------------------------------------------------------------------------------------------
	// Change log table:
	// Version    Date          Expert in charge    Changes applied
	// 01.00.00   07.04.2020    FR                  First release version v1.0
	// 02.00.00   06.12.2022    FR                  Added pointTable
	// 02.00.01   07.02.2023    FR                  Fixed wrong index at pointTable
	// 03.00.00   09.09.2024    FR                  Changed pathData from Variant to "LKinCtrl_typePathData"
	// 03.01.00   17.09.2024    JH                  Do not overwrite coordinate
	//===========================================================================================
	
	// Set return value
	#LKinCtrl_GetPathDataCmd := 16#00;
	
	// Init to avoid warning in point part
	#pathDataCommand.cmdName := '';
	
	// Copy command
	#pathDataCommand := #pathData.commands[#index];
	#parameterValid := #pathDataCommand.parameterValid;
	
	// Check target point
	#tempPoint := #pathDataCommand.point;
	
	// Check if point is used, then copy point coordinates
	IF #tempPoint >= 0 THEN
	  // Check limits
	  IF #tempPoint <= UPPER_BOUND(ARR := #pointTable, DIM := 1)
	    AND #tempPoint >= LOWER_BOUND(ARR := #pointTable, DIM := 1)
	  THEN
	    // Point index is ok
	    // Copy point name to cmd name if no name is provided already
	    IF #pathDataCommand.cmdName = '' THEN
	      #pathDataCommand.cmdName := WSTRING_TO_STRING(#pointTable[#tempPoint].name);
	    END_IF;
	    
	    #pathDataCommand.cmdCoordinates.cartesianPosition.x := #pointTable[#tempPoint].position[0];
	    #pathDataCommand.cmdCoordinates.cartesianPosition.y := #pointTable[#tempPoint].position[1];
	    #pathDataCommand.cmdCoordinates.cartesianPosition.z := #pointTable[#tempPoint].position[2];
	    #pathDataCommand.cmdCoordinates.cartesianPosition.a := #pointTable[#tempPoint].position[3];
	    #pathDataCommand.cmdCoordinates.cartesianPosition.b := #pointTable[#tempPoint].position[4];
	    #pathDataCommand.cmdCoordinates.cartesianPosition.c := #pointTable[#tempPoint].position[5];
	    #pathDataCommand.cmdParameters.moveDirectParameters.linkConstellation := #pointTable[#tempPoint].linkConstellation;
	    #pathDataCommand.cmdParameters.moveDirectParameters.turnJoint := #pointTable[#tempPoint].turnJoint;
	    
	    // do not overwrite coordinate system for set OCS/UCS command
	    IF #pathDataCommand.cmdType <> "LKINCTRL_MC_SET_OCS_FRAME" AND #pathDataCommand.cmdType <> "LKINCTRL_MC_SET_USER_FRAME" THEN
	      #pathDataCommand.cmdCoordinates.coordSystem := #pointTable[#tempPoint].coordSystem;
	    END_IF;
	    
	    FOR #tempCtr := 1 TO "LKINCTRL_NO_OF_VALID_BITS" DO
	      #parameterValid[#tempCtr] := TRUE;
	    END_FOR;
	  ELSE
	    // Invalid point index
	    // Set return value to error
	    #LKinCtrl_GetPathDataCmd := 16#02;
	    RETURN;
	  END_IF;
	ELSE
	  ; // Not used
	END_IF;
	
	
	// Check auxPoint
	#tempPoint := #pathDataCommand.cmdParameters.circleParameters.point;
	
	// Check if aux point is used, then copy point coordinates
	IF #tempPoint >= 0 THEN
	  // Check limits
	  IF #tempPoint <= UPPER_BOUND(ARR := #pointTable, DIM := 1)
	    AND #tempPoint >= LOWER_BOUND(ARR := #pointTable, DIM := 1)
	  THEN
	    ; // Point index is ok
	    #pathDataCommand.cmdParameters.circleParameters.auxPoint[1] := #pointTable[#tempPoint].position[0];
	    #pathDataCommand.cmdParameters.circleParameters.auxPoint[2] := #pointTable[#tempPoint].position[1];
	    #pathDataCommand.cmdParameters.circleParameters.auxPoint[3] := #pointTable[#tempPoint].position[2];
	    
	    // Check if circMode only contains auxPoint then also copy coordinate system
	    IF #pathDataCommand.cmdParameters.circleParameters.circMode = "CM_CENTER" THEN
	      #pathDataCommand.cmdCoordinates.coordSystem := #pointTable[#tempPoint].coordSystem;
	    END_IF;
	    
	  ELSE
	    // Invalid point index
	    // Set return value to error
	    #LKinCtrl_GetPathDataCmd := 16#03;
	    RETURN;
	  END_IF;
	ELSE
	  ; // Not used
	END_IF;
	
	
	
	
	
	
	
	
END_FUNCTION

FUNCTION "LKinCtrl_CheckPathDataCmd" : Word
TITLE = LKinCtrl_CheckPathDataCmd
{ S7_Optimized_Access := 'TRUE' }
AUTHOR : 'handling.team.automation@siemens.com'
FAMILY : LKinCtrl
VERSION : 5.0
//The FC checks a PathData command to be configured correctly
   VAR_INPUT 
      firstFlag : DInt;
      lastFlag : DInt;
      firstValueFlag : DInt;
      lastValueFlag : DInt;
   END_VAR

   VAR_OUTPUT 
      cmdIsMotionCmd : Bool;   // TRUE: Command is a motion command
   END_VAR

   VAR_IN_OUT 
      pathDataCmd : Variant;   // variant for PathData command
   END_VAR

   VAR_TEMP 
      tempFlagCtr : Int;   // temporary counter for flags
      tempPathDataCmd_regular : REF_TO "LKinCtrl_typePathDataElement";   // temporary reference to PathData element
      tempPathDataCmd_PreBuf : REF_TO "LKinCtrl_typePathDataElement_PreBuf";   // temporary reference to PathData_PreBuf element
      tempPathDataCmd_checking : "LKinCtrl_typePathDataElement" := ((), (), (), (), (), (((), (), (), (), (), ()), ()), (((), (), (), ()), ((), (), (), ()), (), (), [-1.0], (), (), ((), (), [()]), ((), ()), (()), ((), (), [()], (), (), (), ()), ((), (), ()), (([()], (), (), ()), ([()], (), (), ()))), [((), (), ()), ((), (), ()), ((), (), ())], [((), (), (), ()), ((), (), (), ()), ((), (), (), ()), ((), (), (), ())], [6(TRUE)]);   // temporary variable for PathDataElement being checked
   END_VAR

   VAR CONSTANT 
      STATUS_NO_ERROR_IN_COMMAND : Word := 16#0000;   // status no error found command
      ERR_PATHDATA_CMDTYPE : Word := 16#80A0;   // error due to wrong cmdType
      ERR_PATHDATA_COORDSYSTEM : Word := 16#80B1;   // error due to wrong coordinate system
      ERR_PATHDATA_VELOCITY : Word := 16#8003;   // error due to wrong velocity
      ERR_PATHDATA_ACCELERATION : Word := 16#8004;   // error due to wrong acceleration
      ERR_PATHDATA_DECELERATION : Word := 16#8005;   // error due to wrong deceleration
      ERR_PATHDATA_JERK : Word := 16#8006;   // error due to wrong jerk
      ERR_PATHDATA_ORIENTATIONDIRECTION : Word := 16#8007;   // error due to wrong orientation direction
      ERR_PATHDATA_BUFFERMODE : Word := 16#80B2;   // error due to wrong buffer mode
      ERR_PATHDATA_DYNAMICADAPTION : Word := 16#80B5;   // error due to wrong dynamic adaption
      ERR_PATHDATA_CIRCMODE : Word := 16#80B6;   // error due to wrong circle mode
      ERR_PATHDATA_PATHCHOICE : Word := 16#80B9;   // error due to wrong path choice
      ERR_PATHDATA_CIRCLEPLANE : Word := 16#80BA;   // error due to wrong circle plane
      ERR_PATHDATA_RADIUS : Word := 16#80BB;   // error due to wrong radius
      ERR_PATHDATA_ARC : Word := 16#80BC;   // error due to wrong arc
      ERR_PATHDATA_SETFLAGS_FLAG : Word := 16#80D1;   // error due to wrong set flag definition
      ERR_PATHDATA_SETFLAGS_FLAGMODE : Word := 16#80D2;   // error due to wrong set flag mode definition
      ERR_PATHDATA_VALUEFLAGS_FLAG : Word := 16#80D3;   // error due to wrong value flag definition
      ERR_PATHDATA_VALUEFLAGS_FLAGMODE : Word := 16#80D4;   // error due to wrong value flag mode definition
      ERR_PATHDATA_OFFSET_PARA_NO : Word := 16#80A1;   // error due to wrong offset parameter set number
      ERR_PATHDATA_OFFSET_MAINPATHPLANE : Word := 16#80A2;   // error due to wrong main path plane
      ERR_PATHDATA_POSITIONMODE : Word := 16#80A3;   // error due to wrong position mode
      ERR_PATHDATA_LINK_CONSTELLATION : Word := 16#80A4;   // error due to wrong link constellation
      ERR_PATHDATA_CONVEYOR_PARA_NO : Word := 16#80A5;   // error due to wrong conveyor parameter set number
      ERR_PATHDATA_TOOLNUMBER : Word := 16#80A6;   // error due to wrong tool number
      ERR_PATHDATA_COORDINATES : Word := 16#80A7;   // error due to wrong coordinates
      ERR_PATHDATA_ZONENUMBER : Word := 16#80A8;   // error due to wrong zone number
      ERR_PATHDATA_ZONECONFIGURATIONINDEX : Word := 16#80A9;   // error due to wrong zone configuration index
      ERR_PATHDATA_ZONEDEACTIVATIONMODE : Word := 16#80AA;   // error due to wrong zone de-/activation mode
      ERR_PATHDATA_PICKANDPLACE_STARTVECTOR : Word := 16#80AB;   // error due to wrong pick and place start vector parametrization
      ERR_PATHDATA_PICKANDPLACE_TARGETVECTOR : Word := 16#80AC;   // error due to wrong pick and place target vector parametrization
      ERR_PATHDATA_PICKANDPLACE_BLENDING_NOT_POSSIBLE : Word := 16#80AD;   // error due to invalid buffer mode
   END_VAR


BEGIN
	//==========================================================================================
	// SIEMENS AG
	// (c)Copyright 2020 All Rights Reserved
	//------------------------------------------------------------------------------------------
	// Library: LKinCtrl
	// Tested with: S7-1517T-3 PN/DP
	// Engineering: TIA Portal V15
	// Restrictions: ---
	// Requirements: S7-1500T FW 2.8
	// Functionality: LKinCtrl_CheckPathDataCmd
	// The FC checks a PathData command to be configured correctly
	//
	// Support: tech.team.motioncontrol@siemens.com
	// Note: Parameter comments are only available in language 'English (United States)'
	//------------------------------------------------------------------------------------------
	// Change log table:
	// Version    Date          Expert in charge    Changes applied
	// 01.00.00   26.02.2019    JR                  First release version v1.0
	// 01.01.00   14.06.2019    JR                  added flagOnly command
	// 01.02.00   03.12.2019    JR                  added command checks for value flags
	// 01.02.01   30.01.2020    FR                  separate constant for flag arrays
	// 01.02.02   09.04.2020    FR                  copy valueFlags & CS to temp also
	// 01.03.00   16.04.2020    FR                  added moveDirect & trackConveyor
	// 01.03.01   14.01.2021    FR                  added check for wait time 
	// 01.04.00   25.01.2021    FR                  added SetFrame cmd and restructured FC
	// 01.04.01   29.10.2021    FR                  allow FM25 & FM26
	// 01.04.02   03.01.2024    SF                  added check for PickAndPlace command
	// 02.00.00   28.10.2024    JH                  removed dependency from _reduced and _advanced path data types
	//===========================================================================================
	
	// FC initialization
	//====================================================================================================================================
	#LKinCtrl_CheckPathDataCmd := #STATUS_NO_ERROR_IN_COMMAND;
	
	// PathData conversion (reduced, regular(no suffix), advanced)
	//===========================================================================================
	REGION PATHDATA_ELEMENT_CONVERSION
	  // regular PathDataCommand
	  IF TypeOf(#pathDataCmd) = "LKinCtrl_typePathDataElement" THEN
	    // reference internal PathDataCommand to attached Variant
	    #tempPathDataCmd_regular ?= #pathDataCmd;
	    // copy to internal PathData (full version)
	    #tempPathDataCmd_checking.cmdType := #tempPathDataCmd_regular^.cmdType;
	    #tempPathDataCmd_checking.cmdCoordinates.cartesianPosition := #tempPathDataCmd_regular^.cmdCoordinates.cartesianPosition;
	    #tempPathDataCmd_checking.cmdCoordinates.coordSystem := #tempPathDataCmd_regular^.cmdCoordinates.coordSystem;
	    #tempPathDataCmd_checking.cmdParameters := #tempPathDataCmd_regular^.cmdParameters;
	    #tempPathDataCmd_checking.setFlags := #tempPathDataCmd_regular^.setFlags;
	    #tempPathDataCmd_checking.valueFlags := #tempPathDataCmd_regular^.valueFlags;
	    
	    // PathDataPreBuffered PathDataCommand
	  ELSIF TypeOf(#pathDataCmd) = "LKinCtrl_typePathDataElement_PreBuf" THEN
	    #tempPathDataCmd_PreBuf ?= #pathDataCmd;
	    // copy to internal PathData (full version)
	    #tempPathDataCmd_checking.cmdType := #tempPathDataCmd_PreBuf^.cmdType;
	    #tempPathDataCmd_checking.cmdCoordinates.cartesianPosition.x := #tempPathDataCmd_PreBuf^.cmdCoordinates.targetPosition[1];
	    #tempPathDataCmd_checking.cmdCoordinates.cartesianPosition.y := #tempPathDataCmd_PreBuf^.cmdCoordinates.targetPosition[2];
	    #tempPathDataCmd_checking.cmdCoordinates.cartesianPosition.z := #tempPathDataCmd_PreBuf^.cmdCoordinates.targetPosition[3];
	    #tempPathDataCmd_checking.cmdCoordinates.cartesianPosition.a := #tempPathDataCmd_PreBuf^.cmdCoordinates.targetPosition[4];
	    #tempPathDataCmd_checking.cmdCoordinates.cartesianPosition.b := #tempPathDataCmd_PreBuf^.cmdCoordinates.targetPosition[5];
	    #tempPathDataCmd_checking.cmdCoordinates.cartesianPosition.c := #tempPathDataCmd_PreBuf^.cmdCoordinates.targetPosition[6];
	    #tempPathDataCmd_checking.cmdCoordinates.coordSystem := #tempPathDataCmd_PreBuf^.cmdCoordinates.coordSystem;
	    #tempPathDataCmd_checking.cmdParameters := #tempPathDataCmd_PreBuf^.cmdParameters;
	    #tempPathDataCmd_checking.setFlags := #tempPathDataCmd_PreBuf^.setFlags;
	    #tempPathDataCmd_checking.valueFlags := #tempPathDataCmd_PreBuf^.valueFlags;
	    
	  //   // advanced PathDataCommand
	  // ELSIF TypeOf(#pathDataCmd) = "LKinCtrl_typePathDataElement_advanced" THEN
	  //   // reference internal PathDataCommand to attached Variant
	  //   #tempPathDataCmd_advanced ?= #pathDataCmd;
	  //   // copy to internal PathData (full version)
	  //   #tempPathDataCmd_checking.cmdType := #tempPathDataCmd_advanced^.cmdType;
	  //   #tempPathDataCmd_checking.cmdCoordinates.cartesianPosition := #tempPathDataCmd_advanced^.cmdCoordinates.cartesianPosition;
	  //   #tempPathDataCmd_checking.cmdCoordinates.coordSystem := #tempPathDataCmd_advanced^.cmdCoordinates.coordSystem;
	  //   #tempPathDataCmd_checking.cmdParameters := #tempPathDataCmd_advanced^.cmdParameters;
	  //   #tempPathDataCmd_checking.setFlags := #tempPathDataCmd_advanced^.setFlags;
	  //   #tempPathDataCmd_checking.valueFlags := #tempPathDataCmd_advanced^.valueFlags;
	    
	  //   // reduced PathDataCommand
	  // ELSIF TypeOf(#pathDataCmd) = "LKinCtrl_typePathDataElement_reduced" THEN
	  //   // reference internal PathDataCommand to attached Variant
	  //   #tempPathDataCmd_reduced ?= #pathDataCmd;
	  //   // copy to internal PathData (full version)
	  //   #tempPathDataCmd_checking.cmdType := #tempPathDataCmd_reduced^.cmdType;
	  //   #tempPathDataCmd_checking.cmdCoordinates.cartesianPosition := #tempPathDataCmd_reduced^.cmdCoordinates.cartesianPosition;
	  //   #tempPathDataCmd_checking.cmdCoordinates.coordSystem := #tempPathDataCmd_reduced^.cmdCoordinates.coordSystem;
	  //   #tempPathDataCmd_checking.cmdParameters.pathDynamics := #tempPathDataCmd_reduced^.cmdParameters.pathDynamics;
	  //   #tempPathDataCmd_checking.cmdParameters.orientationDirection := #tempPathDataCmd_reduced^.cmdParameters.orientationDirection;
	  //   #tempPathDataCmd_checking.cmdParameters.bufferMode := #tempPathDataCmd_reduced^.cmdParameters.bufferMode;
	  //   #tempPathDataCmd_checking.cmdParameters.transitionParameters := #tempPathDataCmd_reduced^.cmdParameters.transitionParameters;
	  //   #tempPathDataCmd_checking.cmdParameters.dynamicAdaption := #tempPathDataCmd_reduced^.cmdParameters.dynamicAdaption;
	  //   #tempPathDataCmd_checking.setFlags := #tempPathDataCmd_reduced^.setFlags;
	  //   #tempPathDataCmd_checking.valueFlags := #tempPathDataCmd_reduced^.valueFlags;
	    
	  ELSE
	    // Invalid data type 
	    RETURN;
	    
	  END_IF;
	END_REGION PATHDATA_CONVERSION 
	
	
	
	
	REGION CHECK_COMMAND
	  // Init motionCmd to false
	  #cmdIsMotionCmd := FALSE;
	  
	  // --------------------------------------------------------
	  // Check settings depending on cmd type
	  // --------------------------------------------------------
	  REGION CMD_SPECIFIC
	    
	    CASE #tempPathDataCmd_checking.cmdType OF
	      "LKINCTRL_CMD_FLAG_ONLY":  // cmdType = 0
	        ;
	        
	      "LKINCTRL_MC_MOVELINEARABS", "LKINCTRL_MC_MOVELINEARREL":  // cmdType = 1,2
	        REGION LINEAR
	          // Set motion cmd to true
	          #cmdIsMotionCmd := TRUE;
	          
	          // Check coordinate system
	          CASE #tempPathDataCmd_checking.cmdCoordinates.coordSystem OF
	            "CS_WCS".."CS_OCS3",  // Regular frames
	            "LKINCTRL_CS_NO_OF_FIRST_USER_FRAME".."LKINCTRL_CS_NO_OF_LAST_USER_FRAME":  // User frames
	              ; // OK -> do nothing
	            ELSE  // Invalid CS for linear command
	              #LKinCtrl_CheckPathDataCmd := #ERR_PATHDATA_COORDSYSTEM;
	              RETURN;
	          END_CASE;
	          
	          // Check dynamics
	          IF #tempPathDataCmd_checking.cmdParameters.pathDynamics.velocity = 0.0 THEN
	            #LKinCtrl_CheckPathDataCmd := #ERR_PATHDATA_VELOCITY;
	            RETURN;
	          END_IF;
	          IF #tempPathDataCmd_checking.cmdParameters.pathDynamics.acceleration = 0.0 THEN
	            #LKinCtrl_CheckPathDataCmd := #ERR_PATHDATA_ACCELERATION;
	            RETURN;
	          END_IF;
	          IF #tempPathDataCmd_checking.cmdParameters.pathDynamics.deceleration = 0.0 THEN
	            #LKinCtrl_CheckPathDataCmd := #ERR_PATHDATA_DECELERATION;
	            RETURN;
	          END_IF;
	        END_REGION
	        
	      "LKINCTRL_MC_MOVECIRCULARABS", "LKINCTRL_MC_MOVECIRCULARREL": // cmdType 3,4
	        REGION CIRCULAR
	          // Set motion cmd to true
	          #cmdIsMotionCmd := TRUE;
	          
	          // Check coordinate system
	          CASE #tempPathDataCmd_checking.cmdCoordinates.coordSystem OF
	            "CS_WCS".."CS_OCS3",  // Regular frames
	            "LKINCTRL_CS_NO_OF_FIRST_USER_FRAME".."LKINCTRL_CS_NO_OF_LAST_USER_FRAME":  // User frames
	              ; // OK -> do nothing
	            ELSE  // Invalid CS for linear command
	              #LKinCtrl_CheckPathDataCmd := #ERR_PATHDATA_COORDSYSTEM;
	              RETURN;
	          END_CASE;
	          
	          // Check dynamics
	          IF #tempPathDataCmd_checking.cmdParameters.pathDynamics.velocity = 0.0 THEN
	            #LKinCtrl_CheckPathDataCmd := #ERR_PATHDATA_VELOCITY;
	            RETURN;
	          END_IF;
	          IF #tempPathDataCmd_checking.cmdParameters.pathDynamics.acceleration = 0.0 THEN
	            #LKinCtrl_CheckPathDataCmd := #ERR_PATHDATA_ACCELERATION;
	            RETURN;
	          END_IF;
	          IF #tempPathDataCmd_checking.cmdParameters.pathDynamics.deceleration = 0.0 THEN
	            #LKinCtrl_CheckPathDataCmd := #ERR_PATHDATA_DECELERATION;
	            RETURN;
	          END_IF;
	          
	          //PathData - command - circleParameter - circMode
	          IF #tempPathDataCmd_checking.cmdParameters.circleParameters.circMode < "CM_BORDER"
	            OR #tempPathDataCmd_checking.cmdParameters.circleParameters.circMode > "LKINCTRL_CIRCMODE_GCODE" //"CM_RADIUS"
	          THEN
	            #LKinCtrl_CheckPathDataCmd := #ERR_PATHDATA_CIRCMODE;
	            RETURN;
	          END_IF;
	          
	          //PathData - command - circleParameter - pathChoice
	          IF #tempPathDataCmd_checking.cmdParameters.circleParameters.pathChoice < "PC_POSITIVE"
	            OR #tempPathDataCmd_checking.cmdParameters.circleParameters.pathChoice > "PC_LONG_RUN_NEGATIVE"
	          THEN
	            #LKinCtrl_CheckPathDataCmd := #ERR_PATHDATA_PATHCHOICE;
	            RETURN;
	          END_IF;
	          
	          //PathData - command - circleParameter - circlePlane
	          IF #tempPathDataCmd_checking.cmdParameters.circleParameters.circlePlane < "CP_XZ"
	            OR #tempPathDataCmd_checking.cmdParameters.circleParameters.circlePlane > "CP_XY"
	          THEN
	            #LKinCtrl_CheckPathDataCmd := #ERR_PATHDATA_CIRCLEPLANE;
	            RETURN;
	          END_IF;
	          
	          //PathData - command - circleParameter - radius
	          IF #tempPathDataCmd_checking.cmdParameters.circleParameters.radius < 0.0 THEN
	            #LKinCtrl_CheckPathDataCmd := #ERR_PATHDATA_RADIUS;
	            RETURN;
	          END_IF;
	          
	          //PathData - command - circleParameter - arc
	          IF #tempPathDataCmd_checking.cmdParameters.circleParameters.arc < 0.0 THEN
	            #LKinCtrl_CheckPathDataCmd := #ERR_PATHDATA_ARC;
	            RETURN;
	          END_IF;
	        END_REGION
	        
	      "LKINCTRL_MC_MOVEDIRECTABS", "LKINCTRL_MC_MOVEDIRECTREL": // cmdType = 5,6
	        REGION MOVE_DIRECT
	          // Set motion cmd to true
	          #cmdIsMotionCmd := TRUE;
	          
	          // Check coordinate system
	          CASE #tempPathDataCmd_checking.cmdCoordinates.coordSystem OF
	            "CS_WCS".."CS_OCS3",  // Regular frames
	            "LKINCTRL_CS_NO_OF_FIRST_USER_FRAME".."LKINCTRL_CS_NO_OF_LAST_USER_FRAME",  // User frames
	            "CS_MCS", // MCS also allowed
	            "CS_JCS": // JCS also allowed
	              ; // OK -> do nothing
	            ELSE  // Invalid CS for linear command
	              #LKinCtrl_CheckPathDataCmd := #ERR_PATHDATA_COORDSYSTEM;
	              RETURN;
	          END_CASE;
	          
	          // Check MoveDirect dynamics
	          IF #tempPathDataCmd_checking.cmdParameters.pathDynamics.velocity > 1.0
	            OR #tempPathDataCmd_checking.cmdParameters.pathDynamics.velocity = 0.0
	          THEN
	            #LKinCtrl_CheckPathDataCmd := #ERR_PATHDATA_VELOCITY;
	            RETURN;
	          END_IF;
	          IF #tempPathDataCmd_checking.cmdParameters.pathDynamics.acceleration > 1.0
	            OR #tempPathDataCmd_checking.cmdParameters.pathDynamics.acceleration = 0.0
	          THEN
	            #LKinCtrl_CheckPathDataCmd := #ERR_PATHDATA_ACCELERATION;
	            RETURN;
	          END_IF;
	          IF #tempPathDataCmd_checking.cmdParameters.pathDynamics.deceleration > 1.0
	            OR #tempPathDataCmd_checking.cmdParameters.pathDynamics.deceleration = 0.0
	          THEN
	            #LKinCtrl_CheckPathDataCmd := #ERR_PATHDATA_DECELERATION;
	            RETURN;
	          END_IF;
	          IF (#tempPathDataCmd_checking.cmdParameters.pathDynamics.jerk > 0.0
	            AND #tempPathDataCmd_checking.cmdParameters.pathDynamics.jerk < 0.1)
	            OR #tempPathDataCmd_checking.cmdParameters.pathDynamics.jerk > 0.9
	          THEN
	            #LKinCtrl_CheckPathDataCmd := #ERR_PATHDATA_JERK;
	            RETURN;
	          END_IF;
	          
	          // PathData - command - moveDirect Parameters - linkConstellation
	          // IF #tempPathDataCmd_checking.cmdParameters.moveDirectParameters.linkConstellation <> 16#FFFF_FFFF
	          //   AND #tempPathDataCmd_checking.cmdParameters.moveDirectParameters.linkConstellation > 16#0000_0007
	          // THEN
	          //   #LKinCtrl_CheckPathDataCmd := #ERR_PATHDATA_LINK_CONSTELLATION;
	          //   RETURN;
	          // END_IF;
	          
	          //PathData - command - moveDirect Parameters - positionMode
	          IF #tempPathDataCmd_checking.cmdParameters.moveDirectParameters.positionMode < "PM_ABS_ABS"
	            OR #tempPathDataCmd_checking.cmdParameters.moveDirectParameters.positionMode > "PM_ABS_REL"
	          THEN
	            #LKinCtrl_CheckPathDataCmd := #ERR_PATHDATA_POSITIONMODE;
	            RETURN;
	          END_IF;
	        END_REGION
	        
	      "LKINCTRL_MC_TRACKCONVEYORBELT": // cmdType = 10
	        REGION TRACK_CONVEYOR
	          //PathData - command - conveyorParameters - conveyorParaNo
	          IF #tempPathDataCmd_checking.cmdParameters.conveyorParameters.conveyorParaNo < 1
	            OR #tempPathDataCmd_checking.cmdParameters.conveyorParameters.conveyorParaNo > "LKINCTRL_NO_OF_CONVEYOR"
	          THEN
	            #LKinCtrl_CheckPathDataCmd := #ERR_PATHDATA_CONVEYOR_PARA_NO;
	            RETURN;
	          END_IF;
	          
	          // Check conveyTracking coordinate system to be OCS1-3
	          IF #tempPathDataCmd_checking.cmdCoordinates.coordSystem < "CS_OCS1"
	            OR #tempPathDataCmd_checking.cmdCoordinates.coordSystem > "CS_OCS3"
	          THEN
	            #LKinCtrl_CheckPathDataCmd := #ERR_PATHDATA_COORDSYSTEM;
	            RETURN;
	          END_IF;
	        END_REGION
	        
	      "LKINCTRL_MC_MOVELINEARPICKANDPLACE": // cmdType = 11
	        REGION LINEAR_PICK_AND_PLACE
	          
	          // Set motion cmd to true
	          #cmdIsMotionCmd := TRUE;
	          
	          // Check conveyor config
	          IF #tempPathDataCmd_checking.cmdParameters.conveyorParameters.conveyorParaNo < 0
	            OR #tempPathDataCmd_checking.cmdParameters.conveyorParameters.conveyorParaNo > "LKINCTRL_NO_OF_CONVEYOR"
	          THEN
	            #LKinCtrl_CheckPathDataCmd := #ERR_PATHDATA_CONVEYOR_PARA_NO;
	            RETURN;
	          END_IF;
	          
	          // Check coordinate system
	          CASE #tempPathDataCmd_checking.cmdCoordinates.coordSystem OF
	            "CS_WCS".."CS_OCS3":  // Regular frames
	              ; // OK -> do nothing
	            ELSE  // Invalid CS for linear command
	              #LKinCtrl_CheckPathDataCmd := #ERR_PATHDATA_COORDSYSTEM;
	              RETURN;
	          END_CASE;
	          
	          // Check dynamics
	          IF #tempPathDataCmd_checking.cmdParameters.pathDynamics.velocity = 0.0
	            OR #tempPathDataCmd_checking.cmdParameters.orientationDynamics.velocity = 0.0
	          THEN
	            #LKinCtrl_CheckPathDataCmd := #ERR_PATHDATA_VELOCITY;
	            RETURN;
	          END_IF;
	          IF #tempPathDataCmd_checking.cmdParameters.pathDynamics.acceleration = 0.0
	            OR #tempPathDataCmd_checking.cmdParameters.orientationDynamics.acceleration = 0.0
	          THEN
	            #LKinCtrl_CheckPathDataCmd := #ERR_PATHDATA_ACCELERATION;
	            RETURN;
	          END_IF;
	          IF #tempPathDataCmd_checking.cmdParameters.pathDynamics.deceleration = 0.0
	            OR #tempPathDataCmd_checking.cmdParameters.orientationDynamics.deceleration = 0.0
	          THEN
	            #LKinCtrl_CheckPathDataCmd := #ERR_PATHDATA_DECELERATION;
	            RETURN;
	          END_IF;
	          
	          //Check if start vector is existent
	          IF NOT (#tempPathDataCmd_checking.cmdParameters.pickAndPlaceParameters.startParameter.direction[1] = 0.0
	            AND #tempPathDataCmd_checking.cmdParameters.pickAndPlaceParameters.startParameter.direction[2] = 0.0
	            AND #tempPathDataCmd_checking.cmdParameters.pickAndPlaceParameters.startParameter.direction[3] = 0.0)
	          THEN
	            //start vector existent
	            //check working heigth and dynamics factor
	            IF #tempPathDataCmd_checking.cmdParameters.pickAndPlaceParameters.startParameter.workingHeight < 0.0 THEN
	              #LKinCtrl_CheckPathDataCmd := #ERR_PATHDATA_PICKANDPLACE_STARTVECTOR;
	              RETURN;
	            END_IF;
	            //Check buffer mode
	            IF #tempPathDataCmd_checking.cmdParameters.bufferMode <> "BM_BUFFERED" THEN
	              #LKinCtrl_CheckPathDataCmd := #ERR_PATHDATA_PICKANDPLACE_BLENDING_NOT_POSSIBLE;
	              RETURN;
	            END_IF;
	          END_IF;
	          //Check if target vector is existent
	          IF NOT (#tempPathDataCmd_checking.cmdParameters.pickAndPlaceParameters.targetParameter.direction[1] = 0.0
	            AND #tempPathDataCmd_checking.cmdParameters.pickAndPlaceParameters.targetParameter.direction[2] = 0.0
	            AND #tempPathDataCmd_checking.cmdParameters.pickAndPlaceParameters.targetParameter.direction[3] = 0.0)
	          THEN
	            //target vector existent
	            //check working heigth and dynamics factor
	            IF #tempPathDataCmd_checking.cmdParameters.pickAndPlaceParameters.targetParameter.workingHeight < 0.0 THEN
	              #LKinCtrl_CheckPathDataCmd := #ERR_PATHDATA_PICKANDPLACE_TARGETVECTOR;
	              RETURN;
	            END_IF;
	          END_IF;
	        END_REGION LINEAR_PICK_AND_PLACE
	        
	      "LKINCTRL_MC_SET_OCS_FRAME": // cmdType = 20
	        REGION SET_OCS_FRAME
	          // Check frame to be a OCS
	          IF (#tempPathDataCmd_checking.cmdCoordinates.coordSystem < "CS_OCS1" // First OCS
	            OR #tempPathDataCmd_checking.cmdCoordinates.coordSystem > "CS_OCS3") // Last OCS
	          THEN
	            #LKinCtrl_CheckPathDataCmd := #ERR_PATHDATA_COORDSYSTEM;
	            RETURN;
	          END_IF;
	        END_REGION
	        
	      "LKINCTRL_MC_SET_USER_FRAME": // cmdType = 21
	        REGION SET_USER_FRAME
	          // Check frame to be a user frame
	          IF (#tempPathDataCmd_checking.cmdCoordinates.coordSystem < "LKINCTRL_CS_NO_OF_FIRST_USER_FRAME" // First user frame
	            OR #tempPathDataCmd_checking.cmdCoordinates.coordSystem > "LKINCTRL_CS_NO_OF_LAST_USER_FRAME") // Last user frame
	          THEN
	            #LKinCtrl_CheckPathDataCmd := #ERR_PATHDATA_COORDSYSTEM;
	            RETURN;
	          END_IF;
	        END_REGION
	        
	    "LKINCTRL_MC_SHIFT_CS_REL": //cmdType 60
	      REGION SHIFT_CS_REL
	        ; // Nothing to check?
	      END_REGION
	      
	    "LKINCTRL_MC_RESET_SHIFT": //cmdType 61
	      REGION RESET_CS_SHIFT
	        ; // Nothing to check?
	      END_REGION
	      
	      "LKINCTRL_MC_ACTIVATE_TOOL": // cmdType = 22
	        REGION SET_TOOL
	          // Check tool number (1..3)
	          IF (#tempPathDataCmd_checking.cmdParameters.toolNumber < 1 // First Tool
	            OR #tempPathDataCmd_checking.cmdParameters.toolNumber > 3) // Last Tool
	          THEN
	            #LKinCtrl_CheckPathDataCmd := #ERR_PATHDATA_TOOLNUMBER;
	            RETURN;
	          END_IF;
	        END_REGION
	        
	      "LKINCTRL_MC_SET_TOOL_FRAME": // cmdType = 23
	        REGION DEFINE_TOOL
	          // Check frame (only X,Y,Z,A allowed) --> B and C allowed in 6D
	          // IF (#tempPathDataCmd_checking.cmdCoordinates.cartesianPosition.b <> 0.0) // B
	          //   OR (#tempPathDataCmd_checking.cmdCoordinates.cartesianPosition.c <> 0.0) // C
	          // THEN
	          //   #LKinCtrl_CheckPathDataCmd := #ERR_PATHDATA_COORDINATES;
	          //   RETURN;
	          // END_IF;
	            ;
	        END_REGION
	        
	        
	      "LKINCTRL_MC_DEFINE_WS_ZONE":
	        REGION DEFINE_WS_ZONE
	          // Check configuration index
	          IF #tempPathDataCmd_checking.cmdParameters.zoneParameters.zoneConfigurationIndex < 1
	            OR #tempPathDataCmd_checking.cmdParameters.zoneParameters.zoneConfigurationIndex > "LKINCTRL_NO_OF_ZONES"
	          THEN
	            #LKinCtrl_CheckPathDataCmd := #ERR_PATHDATA_ZONECONFIGURATIONINDEX;
	            RETURN;
	          END_IF;
	          
	          
	          // Check zone number
	          IF #tempPathDataCmd_checking.cmdParameters.zoneParameters.zoneNumber < 1
	            OR #tempPathDataCmd_checking.cmdParameters.zoneParameters.zoneNumber > 10
	          THEN
	            #LKinCtrl_CheckPathDataCmd := #ERR_PATHDATA_ZONENUMBER;
	            RETURN;
	          END_IF;
	        END_REGION
	        
	      "LKINCTRL_MC_ACTIVATE_WS_ZONE":
	        REGION ACTIVATE_WS_ZONE
	          // Check zone number
	          IF #tempPathDataCmd_checking.cmdParameters.zoneParameters.zoneNumber < 1
	            OR #tempPathDataCmd_checking.cmdParameters.zoneParameters.zoneNumber > 10
	          THEN
	            #LKinCtrl_CheckPathDataCmd := #ERR_PATHDATA_ZONENUMBER;
	            RETURN;
	          END_IF;
	        END_REGION
	        
	      "LKINCTRL_MC_DEACTIVATE_WS_ZONE":
	        REGION DEACTIVATE_WS_ZONE
	          CASE #tempPathDataCmd_checking.cmdParameters.zoneParameters.deactivationMode OF
	            "ZONE_DEACTIVATION_MODE_SPECIFIC": // Set a specific zone to inactive
	              // Check zone number
	              IF #tempPathDataCmd_checking.cmdParameters.zoneParameters.zoneNumber < 1
	                OR #tempPathDataCmd_checking.cmdParameters.zoneParameters.zoneNumber > 10
	              THEN
	                #LKinCtrl_CheckPathDataCmd := #ERR_PATHDATA_ZONENUMBER;
	                RETURN;
	              END_IF;
	              
	            "ZONE_DEACTIVATION_MODE_ALL", // Set all workspace zones to inactive
	            "ZONE_DEACTIVATION_MODE_BLOCKED", // Set all blocked zones to inactive
	            "ZONE_DEACTIVATION_MODE_SIGNAL", // Set all signal zones to inactive
	            "ZONE_DEACTIVATION_MODE_WORKSPACE": // Set workspace to inactive
	              ; // Do not check number
	              
	            ELSE  // Invalid mode
	              #LKinCtrl_CheckPathDataCmd := #ERR_PATHDATA_ZONEDEACTIVATIONMODE;
	              RETURN;
	          END_CASE;
	        END_REGION
	        
	      "LKINCTRL_MC_DEFINE_KIN_ZONE":
	        REGION DEFINE_KIN_ZONE
	          // Check configuration index
	          IF #tempPathDataCmd_checking.cmdParameters.zoneParameters.zoneConfigurationIndex < 1
	            OR #tempPathDataCmd_checking.cmdParameters.zoneParameters.zoneConfigurationIndex > "LKINCTRL_NO_OF_ZONES"
	          THEN
	            #LKinCtrl_CheckPathDataCmd := #ERR_PATHDATA_ZONECONFIGURATIONINDEX;
	            RETURN;
	          END_IF;
	          
	          // Check zone number
	          IF #tempPathDataCmd_checking.cmdParameters.zoneParameters.zoneNumber < 2
	            OR #tempPathDataCmd_checking.cmdParameters.zoneParameters.zoneNumber > 10
	          THEN
	            #LKinCtrl_CheckPathDataCmd := #ERR_PATHDATA_ZONENUMBER;
	            RETURN;
	          END_IF;
	        END_REGION
	        
	      "LKINCTRL_MC_ACTIVATE_KIN_ZONE":
	        REGION ACTIAVTE_KIN_ZONE
	          // Check zone number
	          IF #tempPathDataCmd_checking.cmdParameters.zoneParameters.zoneNumber < 2
	            OR #tempPathDataCmd_checking.cmdParameters.zoneParameters.zoneNumber > 10
	          THEN
	            #LKinCtrl_CheckPathDataCmd := #ERR_PATHDATA_ZONENUMBER;
	            RETURN;
	          END_IF;
	        END_REGION
	        
	      "LKINCTRL_MC_DEACTIVATE_KIN_ZONE":
	        REGION DEACTIVATE_KIN_ZONE
	          CASE #tempPathDataCmd_checking.cmdParameters.zoneParameters.deactivationMode OF
	            "ZONE_DEACTIVATION_MODE_SPECIFIC": // Set a specific zone to inactive
	              // Check zone number
	              IF #tempPathDataCmd_checking.cmdParameters.zoneParameters.zoneNumber < 2
	                OR #tempPathDataCmd_checking.cmdParameters.zoneParameters.zoneNumber > 10
	              THEN
	                #LKinCtrl_CheckPathDataCmd := #ERR_PATHDATA_ZONENUMBER;
	                RETURN;
	              END_IF;
	              
	            "ZONE_DEACTIVATION_MODE_ALL": // Set all zones to inactive
	              ; // Do not check number
	              
	            ELSE  // Invalid mode
	              #LKinCtrl_CheckPathDataCmd := #ERR_PATHDATA_ZONEDEACTIVATIONMODE;
	              RETURN;
	          END_CASE;
	        END_REGION
	        
	      "LKINCTRL_CONFIG_END_OFFSET_COMP": // cmdType = 40
	        ;
	        
	      "LKINCTRL_CONFIG_START_OFFSET_COMP_LEFT", "LKINCTRL_CONFIG_START_OFFSET_COMP_RIGHT": // cmdType = 41,42
	        REGION CONTOUR_OFFSET
	          //PathData - command - offsetParameters - offSetParaNo
	          IF #tempPathDataCmd_checking.cmdParameters.offsetParameters.offsetParaNo < 1
	            OR #tempPathDataCmd_checking.cmdParameters.offsetParameters.offsetParaNo > "LKINCTRL_NO_OF_OFFSETS"
	          THEN
	            #LKinCtrl_CheckPathDataCmd := #ERR_PATHDATA_OFFSET_PARA_NO;
	            RETURN;
	          END_IF;
	          
	          //PathData - command - offsetParameters - mainPathPlane
	          IF #tempPathDataCmd_checking.cmdParameters.offsetParameters.mainPathPlane < "CP_XZ"
	            OR #tempPathDataCmd_checking.cmdParameters.offsetParameters.mainPathPlane > "CP_XY"
	          THEN
	            #LKinCtrl_CheckPathDataCmd := #ERR_PATHDATA_OFFSET_MAINPATHPLANE;
	            RETURN;
	          END_IF;
	        END_REGION CONTOUR_OFFSET
	        
	      "LKINCTRL_CMD_WAIT_TIME": // cmdType = 100
	        REGION WAIT_TIME
	          // Check waitTime to be at least 1ms
	          IF #tempPathDataCmd_checking.cmdParameters.pathDynamics.velocity < 1.0 THEN
	            #LKinCtrl_CheckPathDataCmd := #ERR_PATHDATA_VELOCITY;
	          END_IF;
	        END_REGION WAIT_TIME
	        
	      "LKINCTRL_MC_DESYNC_CONVEYOR":
	        REGION DESYNC_CONVEYOR
	          // Check dynamics
	          IF #tempPathDataCmd_checking.cmdParameters.pathDynamics.velocity = 0.0 THEN
	            #LKinCtrl_CheckPathDataCmd := #ERR_PATHDATA_VELOCITY;
	            RETURN;
	          END_IF;
	          IF #tempPathDataCmd_checking.cmdParameters.pathDynamics.acceleration = 0.0 THEN
	            #LKinCtrl_CheckPathDataCmd := #ERR_PATHDATA_ACCELERATION;
	            RETURN;
	          END_IF;
	          IF #tempPathDataCmd_checking.cmdParameters.pathDynamics.deceleration = 0.0 THEN
	            #LKinCtrl_CheckPathDataCmd := #ERR_PATHDATA_DECELERATION;
	            RETURN;
	          END_IF;
	      END_REGION DESYNC_CONVEYOR
	      
	      
	      
	
	      ELSE  // Wrong cmdType
	        #LKinCtrl_CheckPathDataCmd := #ERR_PATHDATA_CMDTYPE;
	        RETURN;
	    END_CASE;
	    
	  END_REGION
	  
	  // --------------------------------------------------------
	  // Check settings independent of cmd type
	  // --------------------------------------------------------
	  REGION CMD_INDEPENDENT
	    //PathData - command - cmdParameters - orientationDirection
	    IF #tempPathDataCmd_checking.cmdParameters.orientationDirection < "DIRA_POSITIVE"
	      OR #tempPathDataCmd_checking.cmdParameters.orientationDirection > "DIRA_SHORTEST"
	    THEN
	      #LKinCtrl_CheckPathDataCmd := #ERR_PATHDATA_ORIENTATIONDIRECTION;
	      RETURN;
	    END_IF;
	    
